// TwinCAT 3 PLC project SlitterPlc
// ProgramVersion: 3.1.4023.0
// libraries:
//   Tc2_Math, * (Beckhoff Automation GmbH)
//   Tc2_MC2, * (Beckhoff Automation GmbH)
//   Tc2_ModbusSrv, * (Beckhoff Automation GmbH)
//   Tc2_Standard, * (Beckhoff Automation GmbH)
//   Tc2_System, * (Beckhoff Automation GmbH)
//   Tc2_Utilities, * (Beckhoff Automation GmbH)
//   Tc2_XmlDataSrv, * (Beckhoff Automation GmbH)
//   Tc3_EventLogger, * (Beckhoff Automation GmbH)
//   Tc3_Module, * (Beckhoff Automation GmbH)
//   Tc3_PackML_V2, * (Beckhoff Automation GmbH)
//   VisuDialogs, * (System)
// project tree:
//   DUTs/Parameters/ ST_CameraParameters.TcDUT, ST_CutterParameters.TcDUT, ST_EjectorParameters.TcDUT, ST_MandrelParameters.TcDUT
//   DUTs/ ST_CameraData.TcDUT, ST_CameraResults.TcDUT, ST_InspectCommands.TcDUT, ST_ManualCommands.TcDUT, ST_TubeParameters.TcDUT
//   Ellipse/ FB_ComputeFromImage.TcPOU, FB_Ellipse.TcPOU, FB_FourthOrder.TcPOU, FB_SecondOrder.TcPOU
//   / GlobalTextList.TcGTLO, PlcTask.TcTTO, Visualization Manager.TcVMO (not stored), VISU_TASK.TcTTO
//   GVLs/ GVL.TcGVL
//   ITFs/ I_Actuator.TcIO, I_Axis.TcIO, I_Camera.TcIO, I_Frame.TcIO
//   POUs/ FB_Actuator.TcPOU, FB_Axis.TcPOU, FB_Base.TcPOU, FB_Camera.TcPOU, FB_Cutter.TcPOU, FB_Ejector.TcPOU, FB_Frame.TcPOU, FB_Mandrel.TcPOU, FB_Slitter.TcPOU, MAIN.TcPOU
//   VISUs/ Front_Panel.TcVIS, Manual_Inspect.TcVIS, MachineSettings.TcVIS, ManualControl.TcVIS, Manual_Camera.TcVIS, Manual_Camera_Calibration.TcVIS, Manual_Camera_Inspection.TcVIS, Manual_Camera_Inspection_Raw.TcVIS, Manual_Camera_RawData.TcVIS, Manual_Cutter.TcVIS, Manual_Ejector.TcVIS, Manual_Frame.TcVIS, Manual_Mandrel.TcVIS, Manual_Vacuum.TcVIS, Manual_Select_Tube.TcVIS, Settings.TcVIS, SettingsTemplate.TcVIS, Settings_Mandrel.TcVIS, Settings_PassCriteria.TcVIS, Settings_ProductDimensions.TcVIS, Visualization.TcVIS

CONFIGURATION SlitterPlc
    RESOURCE PLC ON TwinCAT3
        TASK PlcTask(INTERVAL := T#10ms, PRIORITY := 20);
        TASK VISU_TASK(INTERVAL := T#200000us, PRIORITY := 30);
        PROGRAM MAIN WITH PlcTask : MAIN;
        PROGRAM VisuElems_Visu_Prg WITH VISU_TASK : VisuElems.Visu_Prg;
    END_RESOURCE
END_CONFIGURATION

// ---- DUTs/Parameters/ST_CameraParameters.TcDUT
TYPE ST_CameraParameters :
STRUCT
	pitchRow	: LREAL; // := 0.0250;
	pitchColumn	: LREAL; //  := 0.0219;
	calibrationDistance	: LREAL; // := 3;
	angle		: LREAL; // := 27.65;
END_STRUCT
END_TYPE

// ---- DUTs/Parameters/ST_CutterParameters.TcDUT
TYPE ST_CutterParameters :
STRUCT
	retractPosition	: LREAL; // := 10;
	cutVelocity	: LREAL; // := 20;
END_STRUCT
END_TYPE

// ---- DUTs/Parameters/ST_EjectorParameters.TcDUT
TYPE ST_EjectorParameters :
STRUCT
	ejectPositionPass 	: LREAL; // := 100;
	ejectPositionHome 	: LREAL; // := 50;
	ejectPositionFail 	: LREAL; // := 0;
	ejectVelocity		: LREAL; // := 20;
END_STRUCT
END_TYPE

// ---- DUTs/Parameters/ST_MandrelParameters.TcDUT
TYPE ST_MandrelParameters :
STRUCT
	loadPositionX	: LREAL; // := -72.5;
	velocityX		: LREAL; // := 10;
	loadPositionY	: LREAL; // := -22;
	velocityY		: LREAL; // := 250;
	spindleVelocity	: LREAL; // := 20;
	spindleOffset	: LREAL; // := -1;
	vacuumVelocity	: LREAL; // := 360;
END_STRUCT
END_TYPE

// ---- DUTs/ST_CameraData.TcDUT
TYPE ST_CameraData :
STRUCT
	CurrentJobID			: WORD;
	ErrorCode				: WORD;
	AcquisitionID			: WORD;
	InspectionID			: WORD;
	InspectionResultCode	: WORD;
	Results					: ST_CameraResults;
END_STRUCT
END_TYPE

// ---- DUTs/ST_CameraResults.TcDUT
TYPE ST_CameraResults :
STRUCT
	Count				: REAL;
	WidthMeasurement	: REAL;
	HeightMeasurement	: REAL;
	LocationInX			: REAL;
	LocationInY			: REAL;
	PatternMatchRow		: REAL;
	PatternMatchColumn 	: REAL;
	PointValueRow		: ARRAY[1..GVL.NumberVisionPoints] OF REAL;
	PointValueColumn	: ARRAY[1..GVL.NumberVisionPoints] OF REAL;
END_STRUCT
END_TYPE

// ---- DUTs/ST_InspectCommands.TcDUT
TYPE ST_InspectCommands :
STRUCT
	IncrementSpindle 	: BOOL;
	DecrementSpindle	: BOOL;
	Inspect				: BOOL;	
	InspectComplete		: BOOL;
END_STRUCT
END_TYPE

// ---- DUTs/ST_ManualCommands.TcDUT
TYPE ST_ManualCommands :
STRUCT
	bCalibrateMandrel		: BOOL;
	bCameraCalibrate		: BOOL;
	bCameraComputePeak		: BOOL;
	bCameraTrigger			: BOOL;
	bCameraInspect			: BOOL;
	bCameraRawData			: BOOL;
	bCameraSelectTube		: BOOL;
	bCutSample				: BOOL;
	bCutterDisable			: BOOL;
	bCutterHome				: BOOL;
	bCutterReset			: BOOL;
	bCutterMoveAbs			: BOOL;
	bEjectAxisEnableToggle	: BOOL;
	bEjectAxisFailPosition	: BOOL;
	bEjectAxisHomePosition	: BOOL;
	bEjectAxisPassPosition	: BOOL;
	bEjectAxisReset			: BOOL;
	bEjectReset				: BOOL;
	bEjectSamplePass		: BOOL;
	bEjectSampleFail		: BOOL;
	bEjectZExtend			: BOOL;
	bEjectZNeutral			: BOOL;
	bEjectZRetract			: BOOL;
	bEjectBlowOff			: BOOL;
	bEjectVacuum			: BOOL;
	bEjectXOff				: BOOL;
	bEjectZOff				: BOOL;
	bLowerMandrel			: BOOL;		
	bMandrelXEnableToggle	: BOOL;
	bMandrelYEnableToggle	: BOOL;
	bMandrelSpindleToggle	: BOOL;
	bMandrelSpindleRotate	: BOOL;
	bMandrelReset			: BOOL;
	bMoveToLoadPosition		: BOOL;
	bMoveToCutPosition		: BOOL;
	bMoveToEjectPosition	: BOOL;
	bMoveToInspectPosition	: BOOL;
	bRaiseMandrel			: BOOL;
	bSaveMandrelParameters	: BOOL;
	bToggleMandrelVacuum	: BOOL;
	bVacuumAxisToggleEnable	: BOOL;
	bVacuumAxisMove			: BOOL;
	bVacuumAxisReset		: BOOL;
END_STRUCT
END_TYPE

// ---- DUTs/ST_TubeParameters.TcDUT
TYPE ST_TubeParameters :
STRUCT
	Index				: INT;
	Description			: STRING;
	ProductName			: STRING;
	Diameter			: LREAL;	// diameter [mm] of tube at top protrusion
	DepthOfPocket		: LREAL;	// cut surface offset from top most surface [mm]
	MinLength			: LREAL;	// criteria: minimum length of an allowable cut length [mm]
	MaxLength			: LREAL;	// criteria: maximum length of an allowable cut length [mm]
	MinHeight			: LREAL;	// criteria: minimum width of blob of cut [mm]
	MaxHeight			: LREAL;	// criteria: maximum width of blob of cut [mm]
	ResultToleranceX	: LREAL;	// criteria: allowable difference from center of tube to center of cut x axis
	ResultToleranceY	: LREAL;	// criteria: allowable difference from center of tube to center of cut y axis
	AdjustmentX			: LREAL;  	// adjustment to add to result in mm before determining pass/fail
	AdjustmentY			: LREAL;	// adjustment to add to result in mm before determining pass/fail
	AdjustmentLength	: LREAL;	// adjustment to add to length result in mm before determining pass/fail	
	CutPositionX		: LREAL;	
	CutPositionY		: LREAL;
	InspectPositionX 	: LREAL;
	InspectPositionY 	: LREAL;
	EjectPositionX		: LREAL;
	EjectPositionY		: LREAL;
	VacPosition			: LREAL;	// vacuum axis position
	VacuumThreshold		: REAL; 	// mmHg to detect presence of tube on mandrel	
	ComputerProgram		: STRING := 'Tube';
END_STRUCT
END_TYPE

// ---- GVLs/GVL.TcGVL
{attribute 'qualified_only'}
VAR_GLOBAL CONSTANT
	NumberVisionPoints	: INT := 20;	// number of points from the camera vision system
	NumberEllipsePoints	: INT := 40; 	// number of ellipse points is 2x number of vision points
	Unknowns			: INT := 5;		// ellipse coefficients
	MaxIterations		: INT := 50;	
	ConvergenceCriteria : LREAL := 0.000000001;	
	CameraIpAddress		: STRING := '192.168.1.2';
	ModbusReadOffset	: WORD := 7000;
	ModbusWriteOffset	: WORD := 2000;
END_VAR

// ---- ITFs/I_Actuator.TcIO
INTERFACE I_Actuator

PROPERTY Error : BOOL
GET
END_GET
SET
END_SET
END_PROPERTY

METHOD Extend : INT
VAR_INPUT
END_VAR
END_METHOD

PROPERTY IsExtended : BOOL
GET
END_GET
END_PROPERTY

PROPERTY IsRetracted : BOOL
GET
END_GET
END_PROPERTY

METHOD Neutral : BOOL
VAR_INPUT
END_VAR
END_METHOD

METHOD Retract : INT
VAR_INPUT
END_VAR
END_METHOD

END_INTERFACE

// ---- ITFs/I_Axis.TcIO
INTERFACE I_Axis

PROPERTY ErrorCode : UDINT
GET
END_GET
END_PROPERTY

METHOD Home : INT
VAR_INPUT
	Execute	: BOOL;
END_VAR
END_METHOD

METHOD MoveAbs : INT
VAR_INPUT
	Execute	: BOOL;
END_VAR
END_METHOD

METHOD MoveRel : INT
VAR_INPUT
	Execute	: BOOL;
END_VAR
END_METHOD

PROPERTY NcToPlc : NCTOPLC_AXIS_REF
GET
END_GET
END_PROPERTY

METHOD Power : BOOL
VAR_INPUT
	Enable	: BOOL;
END_VAR
END_METHOD

METHOD Reset : INT
VAR_INPUT
	Execute	: BOOL;
END_VAR
END_METHOD

PROPERTY SetDistance : LREAL
SET
END_SET
END_PROPERTY

PROPERTY SetPosition : LREAL
SET
END_SET
END_PROPERTY

PROPERTY SetVelocity : LREAL
SET
END_SET
END_PROPERTY

PROPERTY Status : ST_AxisStatus
GET
END_GET
END_PROPERTY

END_INTERFACE

// ---- ITFs/I_Camera.TcIO
INTERFACE I_Camera

METHOD Calibrate : BOOL
VAR_INPUT
END_VAR
END_METHOD

PROPERTY CalibrationDistance : LREAL
GET
END_GET
SET
END_SET
END_PROPERTY

PROPERTY CameraProgram : STRING
GET
END_GET
SET
END_SET
END_PROPERTY

METHOD Compute : INT
VAR_INPUT
	Execute		: BOOL;	
END_VAR
END_METHOD

PROPERTY CutLengthWithOffset : REAL
GET
END_GET
SET
END_SET
END_PROPERTY

PROPERTY DeltaXmmWithOffset : REAL
GET
END_GET
SET
END_SET
END_PROPERTY

PROPERTY DeltaYmmWithOffset : REAL
GET
END_GET
SET
END_SET
END_PROPERTY

PROPERTY Fail : BOOL
GET
END_GET
SET
END_SET
END_PROPERTY

METHOD GetCameraData : INT
VAR_INPUT
END_VAR
END_METHOD

METHOD Inspect : INT
VAR_INPUT
	Execute	: BOOL;
END_VAR
END_METHOD

END_INTERFACE

// ---- ITFs/I_Frame.TcIO
INTERFACE I_Frame

METHOD BlinkGreen : BOOL
VAR_INPUT
END_VAR
END_METHOD

PROPERTY ControlLeft : BOOL
GET
END_GET
END_PROPERTY

PROPERTY ControlRight : BOOL
GET
END_GET
END_PROPERTY

PROPERTY Door1 : BOOL
GET
END_GET
END_PROPERTY

PROPERTY Door2 : BOOL
GET
END_GET
END_PROPERTY

PROPERTY Door3 : BOOL
GET
END_GET
END_PROPERTY

PROPERTY GreenLight : BOOL
GET
END_GET
SET
END_SET
END_PROPERTY

END_INTERFACE

// ---- POUs/MAIN.TcPOU
PROGRAM MAIN
VAR PERSISTENT
	TubeSelection		: ARRAY[1..5] OF ST_TubeParameters; // array of tube parameters saved in memory
END_VAR
VAR
	CutOffValve	AT %Q*	: BOOL;
	Tube				: ST_TubeParameters;		// parameters in use by the machine
	TubeHmi				: ST_TubeParameters;		// parameters to edit in the hmi
	
	TubeIndicator		: ARRAY[1..5] OF BOOL := [TRUE, FALSE, FALSE, FALSE, FALSE];		// indicator as to which tube is in use
	
	fbSlitter			: FB_Slitter;				// object of machine
	Frame				: FB_Frame;	
	eCommand			: Tc3_PackML_V2.E_PMLCommand;
	eModeCommand		: DINT := E_PMLProtectedUnitMode.ePMLProtUnitMode_Production;
	eState				: Tc3_PackML_V2.E_PMLState;
	sState				: STRING;
	eMode				: DINT;

	TONhmi				: TON;
	TONidle				: TON := (PT := T#2M);
	ntStartProcess		: NT_StartProcess;

	bSave				: BOOL;
	bProcessing			: BOOL;
	bFailed				: BOOL;
	bPassed				: BOOL;
	fbWritePersistent	: FB_WritePersistentData;

	i					: INT;
	
	bOperation			: BOOL;
	bManual				: BOOL;
	bProductSettings	: BOOL;
	bMachineSettings	: BOOL;
	hmiStatus			: STRING := 'OK';
	PressureOn			: BOOL;
	PressureOnTon		: TON := (PT := T#10S);
	PressureOffTon		: TON := (PT := T#2s);
	hmiReset			: BOOL;
	bInspect			: BOOL;
	bNoDetect			: BOOL;
	InspectCommands		: ST_InspectCommands;
	
	currentUser: WSTRING;
	actualCurrentUser: WSTRING;
	debug1			: INT;
	debug2			: INT;
	nIndex			: INT;
	j				: INT;
	readTubeParameter	: ST_TubeParameters;
	emptyTubeParameter	: ST_TubeParameters;
	FilesLoaded		: BOOL;
	rTrigWriteFiles	: R_TRIG;
	nWriteFiles		: INT;
	fbXmlSrvRead	: FB_XmlSrvRead;
	fbXmlSrvWrite	: FB_XmlSrvWrite;
	fbMessage		: FB_TcMessage;
	x : INT;
END_VAR
VAR PERSISTENT	
	iBatch				: ULINT;
	iCounter			: ULINT;
	iCountFailed		: UINT;
	hmiBatch			: ULINT;
	CycleCounter		: LREAL;
END_VAR

CutOffValve := TRUE;

// set up the event logger message
IF NOT fbMessage.EqualsToEventEntryEx(stOther := TC_EVENTS.SlitterEvents.TubeParameterChange) THEN
	fbMessage.CreateEx(TC_EVENTS.SlitterEvents.TubeParameterChange, 0);
	fbMessage.ipArguments.Clear();
END_IF

// load the config parameters on start up
A_ReadTubeParameters();

// display the current user
IF currentUser <> VisuElems.CurrentFullUserName THEN
	currentUser := VisuElems.CurrentFullUserName;
END_IF

IF bOperation THEN				// when switching to the Operation page
	bOperation := FALSE;
	FOR i:=1 TO 5 DO
		TubeIndicator[i] := FALSE;
	END_FOR
	TubeIndicator[1] := TRUE;
	Tube := TubeSelection[1];	// set the tube selection to the first tube on entering page
	TubeHmi := Tube;			// write the parameters to the HMI display
END_IF

IF bManual THEN
	bManual := FALSE;
	TubeHmi := Tube;	// write the parameters to the HMI display
						// do not change the selected tube
END_IF

IF bProductSettings THEN
	bProductSettings := FALSE;
	FOR i:=1 TO 5 DO
		TubeIndicator[i] := FALSE;
	END_FOR
	TubeIndicator[1] := TRUE;
	Tube := TubeSelection[1];	// on entering product page select the first tube
	TubeHmi := Tube;			// write the parameters to the HMI display
END_IF

IF bMachineSettings THEN
	bMachineSettings := FALSE;
	TubeHmi := Tube;
END_IF

//A_StartVisualization();
A_PackMlCommands();

// this must be called before the fbSlitter execution
// determines the tube that is selected 
FOR i := 1 TO 5 DO
	IF TubeIndicator[i] THEN
		Tube := TubeSelection[i];
	END_IF
END_FOR

// machine object
fbSlitter(
	eCommand := eCommand,
	eModeCommand := eModeCommand,
	Batch := hmiBatch,
	Tube := Tube,
	TubeHmi := TubeHmi,	// used only for manual commands
	Inspect := bInspect,
	InspectCmd := InspectCommands,
	CounterOut => iCounter,
	CountFailedOut => iCountFailed,
	BatchOut => iBatch,
	eState => eState,
	sState => sState,
	eMode => eMode);

IF eState <> E_PMLState.ePMLState_Undefined THEN
	A_MonitorParameters();
	A_WriteParameters();
END_IF	
A_StatusIndicator();
(*		
FOR i := 1 TO 5 DO
	IF TubeIndicator[i] THEN
		debug2 := debug2 + 1;		
		IF MEMCMP(ADR(Tube), ADR(TubeSelection[i]), SIZEOF(tube)) <> 0 THEN
			TubeHmi := Tube;		
			bSave := TRUE;
			debug1 := debug1 + 1;
		END_IF 
	END_IF
END_FOR
*)

ACTION A_MonitorParameters:
IF MEMCMP(ADR(TubeHmi), ADR(TubeSelection[i]), SIZEOF(TubeHmi)) <> 0 THEN
	IF TubeHmi.AdjustmentLength <> TubeSelection[i].AdjustmentLength THEN
		// Tube {0} Parameter {1} changed from {2} to {3}
		fbMessage.ipArguments.Clear();
		fbMessage.ipArguments.AddInt(i).AddString('AdjustmentLength');
		fbMessage.ipArguments.AddLReal(TubeSelection[i].AdjustmentLength).AddLReal(TubeHmi.AdjustmentLength);
		fbMessage.Send(0);
	END_IF
	IF TubeHmi.AdjustmentX <> TubeSelection[i].AdjustmentX THEN
		fbMessage.ipArguments.Clear();
		fbMessage.ipArguments.AddInt(i).AddString('AdjustmentX');
		fbMessage.ipArguments.AddLReal(TubeSelection[i].AdjustmentX).AddLReal(TubeHmi.AdjustmentX);
		fbMessage.Send(0);				
	END_IF
	IF TubeHmi.AdjustmentY <> TubeSelection[i].AdjustmentY THEN
		fbMessage.ipArguments.Clear();
		fbMessage.ipArguments.AddInt(i).AddString('AdjustmentY');
		fbMessage.ipArguments.AddLReal(TubeSelection[i].AdjustmentY).AddLReal(TubeHmi.AdjustmentY);
		fbMessage.Send(0);								
	END_IF
	IF TubeHmi.CutPositionX <> TubeSelection[i].CutPositionX THEN
		fbMessage.ipArguments.Clear();
		fbMessage.ipArguments.AddInt(i).AddString('CutPositionX');
		fbMessage.ipArguments.AddLReal(TubeSelection[i].CutPositionX).AddLReal(TubeHmi.CutPositionX);
		fbMessage.Send(0);												
	END_IF
	IF TubeHmi.CutPositionY <> TubeSelection[i].CutPositionY THEN
		fbMessage.ipArguments.Clear();
		fbMessage.ipArguments.AddInt(i).AddString('CutPositionY');
		fbMessage.ipArguments.AddLReal(TubeSelection[i].CutPositionY).AddLReal(TubeHmi.CutPositionY);
		fbMessage.Send(0);																
	END_IF
	IF TubeHmi.DepthOfPocket <> TubeSelection[i].DepthOfPocket THEN
		fbMessage.ipArguments.Clear();
		fbMessage.ipArguments.AddInt(i).AddString('DepthOfPocket');
		fbMessage.ipArguments.AddLReal(TubeSelection[i].DepthOfPocket).AddLReal(TubeHmi.DepthOfPocket);
		fbMessage.Send(0);																				
	END_IF
	IF TubeHmi.Description <> TubeSelection[i].Description THEN
		fbMessage.ipArguments.Clear();
		fbMessage.ipArguments.AddInt(i).AddString('Description');
		fbMessage.ipArguments.AddString(TubeSelection[i].Description).AddStringByValue(TubeHmi.Description);
		fbMessage.Send(0);																								
	END_IF
	IF TubeHmi.Diameter <> TubeSelection[i].Diameter THEN
		fbMessage.ipArguments.Clear();
		fbMessage.ipArguments.AddInt(i).AddString('Diameter');
		fbMessage.ipArguments.AddLReal(TubeSelection[i].Diameter).AddLReal(TubeHmi.Diameter);
		fbMessage.Send(0);																												
	END_IF
	IF TubeHmi.EjectPositionX <> TubeSelection[i].EjectPositionX THEN
		fbMessage.ipArguments.Clear();
		fbMessage.ipArguments.AddInt(i).AddString('EjectPositionX');
		fbMessage.ipArguments.AddLReal(TubeSelection[i].EjectPositionX).AddLReal(TubeHmi.EjectPositionX);
		fbMessage.Send(0);																												
	END_IF	
	IF TubeHmi.EjectPositionY <> TubeSelection[i].EjectPositionY THEN
		fbMessage.ipArguments.Clear();
		fbMessage.ipArguments.AddInt(i).AddString('EjectPositionY');
		fbMessage.ipArguments.AddLReal(TubeSelection[i].EjectPositionY).AddLReal(TubeHmi.EjectPositionY);
		fbMessage.Send(0);																												
	END_IF
	IF TubeHmi.InspectPositionX <> TubeSelection[i].InspectPositionX THEN
		fbMessage.ipArguments.Clear();
		fbMessage.ipArguments.AddInt(i).AddString('InspectPositionX');
		fbMessage.ipArguments.AddLReal(TubeSelection[i].InspectPositionX).AddLReal(TubeHmi.InspectPositionX);
		fbMessage.Send(0);																																
	END_IF
	IF TubeHmi.InspectPositionY <> TubeSelection[i].InspectPositionY THEN
		fbMessage.ipArguments.Clear();
		fbMessage.ipArguments.AddInt(i).AddString('InspectPositionY');
		fbMessage.ipArguments.AddLReal(TubeSelection[i].InspectPositionY).AddLReal(TubeHmi.InspectPositionY);
		fbMessage.Send(0);																																				
	END_IF
	IF TubeHmi.MaxHeight <> TubeSelection[i].MaxHeight THEN
		fbMessage.ipArguments.Clear();
		fbMessage.ipArguments.AddInt(i).AddString('MaxHeight');
		fbMessage.ipArguments.AddLReal(TubeSelection[i].MaxHeight).AddLReal(TubeHmi.MaxHeight);
		fbMessage.Send(0);																																								
	END_IF
	IF TubeHmi.MaxLength <> TubeSelection[i].MaxLength THEN
		fbMessage.ipArguments.Clear();
		fbMessage.ipArguments.AddInt(i).AddString('MaxLength');
		fbMessage.ipArguments.AddLReal(TubeSelection[i].MaxLength).AddLReal(TubeHmi.MaxLength);
		fbMessage.Send(0);																																												
	END_IF
	IF TubeHmi.MinHeight <> TubeSelection[i].MinHeight THEN
		fbMessage.ipArguments.Clear();
		fbMessage.ipArguments.AddInt(i).AddString('MinHeight');
		fbMessage.ipArguments.AddLReal(TubeSelection[i].MinHeight).AddLReal(TubeHmi.MinHeight);
		fbMessage.Send(0);																																																
	END_IF
	IF TubeHmi.MinLength <> TubeSelection[i].MinLength THEN
		fbMessage.ipArguments.Clear();
		fbMessage.ipArguments.AddInt(i).AddString('MinLength');
		fbMessage.ipArguments.AddLReal(TubeSelection[i].MinLength).AddLReal(TubeHmi.MinLength);
		fbMessage.Send(0);																																																				
	END_IF
	IF TubeHmi.ProductName <> TubeSelection[i].ProductName THEN
		fbMessage.ipArguments.Clear();
		fbMessage.ipArguments.AddInt(i).AddString('ProductName');
		fbMessage.ipArguments.AddString(TubeSelection[i].ProductName).AddString(TubeHmi.ProductName);
		fbMessage.Send(0);																																																				
	END_IF
	IF TubeHmi.ResultToleranceX <> TubeSelection[i].ResultToleranceX THEN
		fbMessage.ipArguments.Clear();
		fbMessage.ipArguments.AddInt(i).AddString('ResultToleranceX');
		fbMessage.ipArguments.AddLReal(TubeSelection[i].ResultToleranceX).AddLReal(TubeHmi.ResultToleranceX);
		fbMessage.Send(0);																																																				
	END_IF
	IF TubeHmi.ResultToleranceY <> TubeSelection[i].ResultToleranceY THEN
		fbMessage.ipArguments.Clear();
		fbMessage.ipArguments.AddInt(i).AddString('ResultToleranceY');
		fbMessage.ipArguments.AddLReal(TubeSelection[i].ResultToleranceY).AddLReal(TubeHmi.ResultToleranceY);
		fbMessage.Send(0);																																																								
	END_IF
	IF TubeHmi.VacuumThreshold <> TubeSelection[i].VacuumThreshold THEN
		fbMessage.ipArguments.Clear();
		fbMessage.ipArguments.AddInt(i).AddString('VacuumThreshold');
		fbMessage.ipArguments.AddLReal(TubeSelection[i].VacuumThreshold).AddLReal(TubeHmi.VacuumThreshold);
		fbMessage.Send(0);																																																								
	END_IF
END_IF
END_ACTION

ACTION A_PackMlCommands:
PressureOffTon(IN := frame.Pressure < 80);
IF PressureOffTon.Q THEN
	PressureOn := FALSE;
END_IF
PressureOnTON(IN := frame.Pressure > 80);
IF PressureOnTON.Q THEN
	PressureOn := TRUE;
END_IF

// pack ml commands
IF (NOT PressureOn OR hmiReset) AND FilesLoaded THEN
 	eCommand := E_PMLCommand.ePMLCommand_Abort;
	hmiReset := FALSE;
	IF NOT PressureOn THEN
		hmiStatus := 'Pressure<80PSIG';
	END_IF
ELSIF eMode = E_PMLProtectedUnitMode.ePMLProtUnitMode_Manual THEN
	hmiStatus := 'Manual Mode';
	IF eModeCommand = E_PMLProtectedUnitMode.ePMLProtUnitMode_Production THEN
		eCommand := E_PMLCommand.ePMLCommand_Abort;
		Frame.GreenLight := FALSE;
	ELSE
		CASE eState OF
			E_PMLState.ePMLState_Undefined: eCommand := E_PMLCommand.ePMLCommand_Abort;
			E_PMLState.ePMLState_Aborted: eCommand := E_PMLCommand.ePMLCommand_Clear;
			E_PMLState.ePMLState_Idle: eCommand := E_PMLCommand.ePMLCommand_Start;
			E_PMLState.ePMLState_Stopped: eCommand := E_PMLCommand.ePMLCommand_Reset;
			E_PMLState.ePMLState_Aborting: eCommand := E_PMLCommand.ePMLCommand_Undefined;
		END_CASE
	END_IF
ELSIF eMode = E_PMLProtectedUnitMode.ePMLProtUnitMode_Production THEN
	hmiStatus := 'Automatic Mode';
	IF eModeCommand = E_PMLProtectedUnitMode.ePMLProtUnitMode_Manual THEN
		eCommand := E_PMLCommand.ePMLCommand_Abort;
	ELSE
		CASE eState OF
			E_PMLState.ePMLState_Undefined:
				IF FilesLoaded THEN
					eCommand := E_PMLCommand.ePMLCommand_Abort;
				END_IF
			E_PMLState.ePMLState_Aborted:  
				//IF NOT Frame.Door1 AND NOT Frame.Door2 THEN
					eCommand := E_PMLCommand.ePMLCommand_Clear;
				//END_IF
			E_PMLState.ePMLState_Idle:
					Frame.GreenLight := Frame.Door1 AND Frame.Door2 AND Frame.Door3 AND Frame.Door4;
					IF Frame.GreenLight THEN
						hmiStatus := 'Ready';
					ELSE
						hmiStatus := 'Door Open';
					END_IF
					IF (Frame.ControlLeft AND Frame.ControlRight) AND Frame.GreenLight THEN
						eCommand := E_PMLCommand.ePMLCommand_Start;
						Frame.GreenLight := FALSE;
					END_IF
			E_PMLState.ePMLState_Complete: eCommand := E_PMLCommand.ePMLCommand_Reset;
														
			E_PMLState.ePMLState_Stopped: eCommand := E_PMLCommand.ePMLCommand_Reset;
			E_PMLState.ePMLState_Aborting: eCommand := E_PMLCommand.ePMLCommand_Undefined;			
		END_CASE
	END_IF
END_IF
END_ACTION

ACTION A_ReadTubeParameters:
x := x + 1;

CASE nIndex OF
	0: // read the info from the config file for the camera
		j := 1;
		nIndex := 10;
	10: // 
		fbXmlSrvRead.sXPath := CONCAT('/Configuration/TubeParameters/Tube', INT_TO_STRING(j));
		fbXmlSrvRead.pSymAddr := ADR(readTubeParameter);
		fbXmlSrvRead.cbSymSize := SIZEOF(readTubeParameter);
		fbXmlSrvRead.bExecute := TRUE;
		nIndex := 20;
	20: // wait for the info to load
		IF NOT fbXmlSrvRead.bBusy THEN
			fbXmlSrvRead.bExecute := FALSE;
			MEMCPY(ADR(TubeSelection[j]), ADR(readTubeParameter), SIZEOF(readTubeParameter));
			MEMCPY(ADR(readTubeParameter), ADR(emptyTubeParameter), SIZEOF(emptyTubeParameter));
			nIndex := 30;
			IF j >= 5 THEN
				nIndex := 30;
			ELSE
				nIndex := 10;
				j := j + 1;
			END_IF
		END_IF
	30: // set variables
		Tube := TubeSelection[1];
		TubeHmi := TubeSelection[1];
		TubeIndicator[1] := TRUE;
		bProcessing := FALSE;
		bPassed := FALSE;
		bFailed := FALSE;
		bNoDetect := FALSE;
		nIndex := 40;
	40: // wait here for files loaded
		IF fbSlitter.ReadParameters(Execute := TRUE) THEN
			fbSlitter.ReadParameters(Execute := FALSE);
			FilesLoaded := TRUE;
			nIndex := 50;
		END_IF
	50: // 
		
END_CASE

fbXmlSrvRead(
	sNetId:= '', 
	ePath:= E_OpenPath.PATH_GENERIC, 
	nMode:= XMLSRV_SKIPMISSING, 
	sFilePath:= 'C:\Configuration.xml');
END_ACTION

ACTION A_StartVisualization:
// start the hmi

TONhmi(IN := TRUE, PT := T#4S);
IF TONhmi.Q THEN
	ntStartProcess(
		NETID := '',
		PATHSTR := 'C:\TwinCAT\3.1\Components\Plc\Tc3PlcHmi\Tc3PlcHmi.exe',
		DIRNAME := 'C:\TwinCAT\3.1\Components\Plc\Tc3PlcHmi\',
		COMNDLINE := 'Tc3PlcHmi.exe',
		START := TRUE);
END_IF
END_ACTION

ACTION A_StatusIndicator:
// status indicator

IF eMode = E_PMLProtectedUnitMode.ePMLProtUnitMode_Production THEN
	CASE fbSlitter.Status OF
		0: // idle if idle is on for more than 2 minutes, remove the result
			TONidle(IN := TRUE);
			bProcessing := FALSE;
			IF TONidle.Q THEN
				bFailed := FALSE;
				bPassed := FALSE;	
				bNoDetect := FALSE;		
			END_IF
		1: // processing
			bProcessing := TRUE;
			bFailed := FALSE;
			bPassed := FALSE;
			bNoDetect := FALSE;
			TONidle(IN := FALSE);
		2: // pass
			bPassed := TRUE;
			bFailed := FALSE;
			bProcessing := FALSE;
			bNoDetect := FALSE;
		3: // fail	
			bPassed := FALSE;
			bFailed := TRUE;
			bProcessing := FALSE;
			bNoDetect := FALSE;
		4: // failed to detect
			bPassed := FALSE;
			bFailed := FALSE;
			bProcessing := FALSE;
			bNoDetect := TRUE;		
	END_CASE
ELSE
	bPassed := FALSE;
	bFailed := FALSE;
	bProcessing := FALSE;
END_IF
END_ACTION

ACTION A_WriteParameters:
// write persistent data 
rTrigWriteFiles(CLK := bSave);
IF rTrigWriteFiles.Q THEN
	fbSlitter.SaveParameters(Execute := FALSE);
	nWriteFiles := 10;
END_IF

IF NOT bSave THEN
	nWriteFiles := 0;
END_IF

CASE nWriteFiles OF
	10: // get the tube into memory
		FOR i := 1 TO 5 DO
			IF TubeIndicator[i] THEN
				A_MonitorParameters();
				TubeSelection[i] := TubeHmi;
				TubeSelection[i].Index := i;
			END_IF
		END_FOR
		j := 1;
		nWriteFiles := 20;
	20: // write the tube parameters
		MEMCPY(ADR(readTubeParameter), ADR(TubeSelection[j]), SIZEOF(readTubeParameter));
		fbXmlSrvWrite.bExecute := TRUE;
		fbXmlSrvWrite.cbSymSize := SIZEOF(readTubeParameter);
		fbXmlSrvWrite.pSymAddr := ADR(readTubeParameter);
		fbXmlSrvWrite.sXPath := CONCAT('/Configuration/TubeParameters/Tube', INT_TO_STRING(j));
		nWriteFiles := 30;
	30: // wait to complete
		IF NOT fbXmlSrvWrite.bBusy THEN
			fbXmlSrvWrite.bExecute := FALSE;
			IF j >= 5 THEN
				nWriteFiles := 40;
			ELSE
				j := j + 1;
				nWriteFiles := 20;
			END_IF
		END_IF
	40: // command slitter to save parameters
		IF fbSlitter.SaveParameters(Execute := TRUE) THEN
			fbSlitter.SaveParameters(Execute := FALSE);
			nWriteFiles := 50;
		END_IF
	50: // done state
		bSave := FALSE;
END_CASE

fbXmlSrvWrite(
	sNetId:= '', 
	ePath:= E_OpenPath.PATH_GENERIC, 
	nMode:= XMLSRV_SKIPMISSING, 
	sFilePath:= 'C:\Configuration.xml');
END_ACTION

END_PROGRAM

// ---- POUs/FB_Slitter.TcPOU
FUNCTION_BLOCK FB_Slitter EXTENDS FB_BASE IMPLEMENTS I_UnitState
VAR_INPUT
	Batch		: ULINT;
	Inspect		: BOOL;					// run routine without cut; just inspect
	InspectCmd	: ST_InspectCommands;
	TubeHmi		: ST_TubeParameters;	// used for manual commands
END_VAR
VAR_IN_OUT
	Tube		: ST_TubeParameters;
END_VAR
VAR_OUTPUT 
	FilesLoaded		: BOOL;
	BatchOut		: ULINT;
	CounterOut		: ULINT;
	CountFailedOut	: UINT;
	Status			: INT; 	// 0 = idle, 1 = processing, 2 = pass, 3 = fail, 4 = no detect
END_VAR
VAR
	Mandrel				: FB_Mandrel;
	MandrelParameters	: ST_MandrelParameters;
	Camera				: FB_Camera;
	CameraParameters	: ST_CameraParameters;
	Cutter				: FB_Cutter;
	CutterParameters 	: ST_CutterParameters;
	Ejector				: FB_Ejector;
	EjectorParameters	: ST_EjectorParameters;
	EjectState			: INT;
	Eject				: BOOL;
	
	Manual		: ST_ManualCommands;
	bBusy		: BOOL;	
	bCalibration: BOOL;
	strJobName	: STRING;	// for manual override of which camera program is used
	nIndex		: INT;
	PreviousTubeIndex	: INT;
	fbFileOpen	: FB_FileOpen;
	fbFileWrite	: FB_FileWrite;
	fbFileClose	: FB_FileClose;
	fbLocalSystemTime	: FB_LocalSystemTime;
	bDecrementSpindle: BOOL;
	bIncrementSpindle: BOOL;
	bInspect: BOOL;
	bInspectComplete: BOOL;
	nCalibrationCounter : INT;
	CalibrationArrayX	: ARRAY[0..CalMax] OF LREAL;
	CalibrationArrayY	: ARRAY[0..CalMax] OF LREAL;
	AverageX 			: LREAL;
	AverageY 			: LREAL;
	
	fbXmlSrvRead		: FB_XmlSrvRead;
	fbXmlSrvWrite		: FB_XmlSrvWrite;

	fbMessageSaved		: FB_TcMessage;
		
END_VAR
VAR CONSTANT
	CalMax	: INT := 9;
END_VAR
VAR PERSISTENT
	Counter		: UINT;
	CountFailed	: UINT;
END_VAR


SUPER^();

IF eState <> E_PMLState.ePMLState_Undefined THEN
	Mandrel.MonitorParameters();
	Camera.MonitorParameters();
	Cutter.MonitorParameters();
	Ejector.MonitorParameters();
END_IF

Mandrel.ConvertVaccum();
Mandrel.TubeParameters := Tube;

IF Batch <> BatchOut THEN
	BatchOut := Batch;
	Counter := 0;
	CountFailed := 0;
END_IF

CounterOut := Counter;
CountFailedOut := CountFailed;

Camera.TubeParameters := Tube;

CASE eState OF
	E_PMLState.ePMLState_Idle: Status := 0;
	E_PMLState.ePMLState_Starting: Status := 1;
	(* put in executing to get fast answer - don't wait for execute to finish
	E_PMLState.ePMLState_Completing:
		IF Camera.Pass THEN
			Status := 2;
		ELSIF Camera.Fail THEN
			Status := 3;
		ELSIF ...
			Status := 4;
		END_IF
	*)
END_CASE

METHOD FB_init : BOOL
VAR_INPUT
	bInitRetains : BOOL; // if TRUE, the retain variables are initialized (warm start / cold start)
	bInCopyCode : BOOL;  // if TRUE, the instance afterwards gets moved into the copy code (online change)
END_VAR
IF NOT fbMessageSaved.EqualsToEventEntryEx(stOther := TC_EVENTS.SlitterEvents.ParametersSaved) THEN
	fbMessageSaved.CreateEx(TC_EVENTS.SlitterEvents.ParametersSaved, 0);
END_IF
END_METHOD

METHOD M_Aborting
M_StateComplete();

bBusy := FALSE;
bCalibration := FALSE;
Cutter.Abort();
Ejector.Abort();
Mandrel.Abort();
M_CalibrateCamera(Execute := FALSE);
Eject := FALSE;
EjectState := 0;
nCalibrationCounter := 0;

Manual.bCameraCalibrate := FALSE;
Manual.bCameraComputePeak := FALSE;
Manual.bCameraInspect := FALSE;
Manual.bCameraRawData := FALSE;
Manual.bCameraTrigger := FALSE;
Manual.bCutSample := FALSE;
Manual.bCutterDisable := FALSE;
Manual.bCutterHome := FALSE;
Manual.bCutterMoveAbs := FALSE;
Manual.bCutterReset := FALSE;
Manual.bEjectAxisEnableToggle := FALSE;
Manual.bEjectAxisFailPosition := FALSE;
Manual.bEjectAxisHomePosition := FALSE;
Manual.bEjectAxisPassPosition := FALSE;
Manual.bEjectAxisReset := FALSE;
Manual.bEjectBlowOff := FALSE;
Manual.bEjectReset := FALSE;
Manual.bEjectSamplePass := FALSE;
Manual.bEjectSampleFail := FALSE;
Manual.bEjectVacuum := FALSE;
Manual.bEjectZExtend := FALSE;
Manual.bEjectZNeutral := FALSE;
Manual.bEjectZOff := FALSE;
Manual.bEjectZRetract := FALSE;
Manual.bLowerMandrel := FALSE;
Manual.bMandrelReset := FALSE;
Manual.bMandrelSpindleRotate := FALSE;
Manual.bMandrelSpindleToggle := FALSE;
Manual.bMandrelXEnableToggle := FALSE;
Manual.bMandrelYEnableToggle := FALSE;
Manual.bMoveToCutPosition := FALSE;
Manual.bMoveToEjectPosition := FALSE;
Manual.bMoveToInspectPosition := FALSE;
Manual.bMoveToLoadPosition := FALSE;
Manual.bRaiseMandrel := FALSE;
Manual.bSaveMandrelParameters := FALSE;
Manual.bToggleMandrelVacuum := FALSE;
Manual.bVacuumAxisToggleEnable := FALSE;
Manual.bVacuumAxisMove := FALSE;
Manual.bVacuumAxisReset := FALSE;
END_METHOD

METHOD M_CalibrateCamera : INT;
VAR_INPUT
	Execute			: BOOL;
END_VAR
VAR_INST
	rTrig			: R_TRIG;
	nIndex			: INT;
	Position		: LREAL;
	debug			: INT;
	debug1			: INT;
	debug2			: INT;
END_VAR
rTrig(CLK := Execute);
IF rTrig.Q THEN
	nIndex := 10;
	Mandrel.MoveToInspectPosition(Execute := FALSE, InspectPositionX := Tube.InspectPositionX, InspectPositionY := Tube.InspectPositionY);
	Mandrel.MoveToLoadPosition(Execute := FALSE);
	Mandrel.MoveXAbs(Execute := FALSE, Position := 0);
	Mandrel.MoveYAbs(Execute := FALSE, Position := 0);
	Camera.TriggerCamera(Execute := FALSE);
	bCalibration := TRUE;
END_IF

IF NOT Execute THEN
	debug := debug + 1;
	nIndex := 0;
END_IF

CASE nIndex OF
	0: // idle state
		M_CalibrateCamera := 0;
		bCalibration := FALSE;
	10: // move to first inspection position
		IF Mandrel.MoveToInspectPosition(Execute := TRUE, InspectPositionX := Tube.InspectPositionX, InspectPositionY := Tube.InspectPositionY) = 1 THEN
			Mandrel.MoveToInspectPosition(Execute := FALSE, InspectPositionX := Tube.InspectPositionX, InspectPositionY := Tube.InspectPositionY);
			nIndex := 20;
		ELSIF Mandrel.MoveToInspectPosition(Execute := TRUE, InspectPositionX := Tube.InspectPositionX, InspectPositionY := Tube.InspectPositionY) = -1 THEN
			Mandrel.MoveToInspectPosition(Execute := FALSE, InspectPositionX := Tube.InspectPositionX, InspectPositionY := Tube.InspectPositionY);
			nIndex := 100;
		END_IF
	20: // trigger the camera
		IF Camera.TriggerCamera(Execute := TRUE) THEN
			Camera.PatternX1 := Camera.PatternMatchX;
			Camera.PatternY1 := Camera.PatternMatchY;
			Camera.TriggerCamera(Execute := FALSE);
			nIndex := 30;
		END_IF
	30: // move to second position in x
		Position := Tube.InspectPositionX + Camera.CalibrationDistance; 
		IF Mandrel.MoveXAbs(Execute := TRUE, Position := Position) = 1 THEN
			Mandrel.MoveXAbs(Execute := FALSE, Position := Position);
			nIndex := 40;
		ELSIF Mandrel.MoveXAbs(Execute := TRUE, Position := Position) = -1 THEN
			Mandrel.MoveXAbs(Execute := FALSE, Position := Position);
			nIndex := 100;
		END_IF
	40: // trigger the camera
		IF Camera.TriggerCamera(Execute := TRUE) THEN
			Camera.PatternX2 := Camera.PatternMatchX;
			Camera.PatternY2 := Camera.PatternMatchY;
			Camera.TriggerCamera(Execute := FALSE);
			nIndex := 50;
		END_IF
	45: // 
		Mandrel.MoveYAbs(Execute := FALSE, Position := 0);
		nIndex := 50;
	50: // move to the third position in y
		Position := Tube.InspectPositionY + Camera.CalibrationDistance; 
		IF Mandrel.MoveYAbs(Execute := TRUE, Position := Position) = 1 THEN
			Mandrel.MoveYAbs(Execute := FALSE, Position := Position);
			nIndex := 60;
		ELSIF Mandrel.MoveYAbs(Execute := TRUE, Position := Position) = -1 THEN
			Mandrel.MoveYAbs(Execute := FALSE, Position := Position);
			nIndex := 100;
		END_IF
	60: // trigger camera
		IF Camera.TriggerCamera(Execute := TRUE) THEN
			Camera.PatternX3 := Camera.PatternMatchX;
			Camera.PatternY3 := Camera.PatternMatchY;
			Camera.TriggerCamera(Execute := FALSE);
			nIndex := 70;
		END_IF
	70: // Calculate the pitch
		Camera.Calibrate();
		nIndex := 80; 
	80: // return to load position	
		IF Mandrel.MoveToLoadPosition(Execute := TRUE) <> 0 THEN
			Mandrel.MoveToLoadPosition(Execute := FALSE);
			nIndex := 90;
		END_IF
	90: // done state
		M_CalibrateCamera := 1;
	 
	100: // error state
		M_CalibrateCamera := -1;
	
END_CASE
END_METHOD

METHOD M_Clearing
CASE eMode OF
	E_PMLProtectedUnitMode.ePMLProtUnitMode_Manual: M_ClearingManual();
	
	E_PMLProtectedUnitMode.ePMLProtUnitMode_Production: M_ClearingProduction();
END_CASE
END_METHOD

METHOD M_ClearingManual : BOOL
VAR_INPUT
END_VAR
M_StateComplete();
//M_ClearingManual := TRUE;
END_METHOD

METHOD M_ClearingProduction : BOOL
VAR_INPUT
END_VAR
CASE nState OF
	0:	// reset the variables
		Mandrel.Clear(Execute := FALSE);
		Cutter.Clear(Execute := FALSE);
		Ejector.Reset(Execute := FALSE);
		nState := 10;
	10: // reset the cutter
		IF Cutter.Clear(Execute := TRUE) = 1 THEN
			Cutter.Clear(Execute := FALSE);
			nState := 20;
		END_IF	
	20: // reset the ejector
		IF Ejector.Reset(Execute := TRUE) = 1 THEN
			Ejector.Reset(Execute := FALSE);
			nState := 30;		END_IF

	30: // reset the different objects
		IF Mandrel.Clear(Execute := TRUE) = 1 THEN
			Mandrel.Clear(Execute := FALSE);
			nState := 40;
		END_IF
	40:	// done state
		M_StateComplete();
END_CASE
END_METHOD


METHOD M_Complete
END_METHOD

METHOD M_Completing

VAR
	EjectSample: INT;
END_VAR
IF eMode = E_PMLProtectedUnitMode.ePMLProtUnitMode_Production THEN
	CASE EjectState OF
		0: // wait for eject command
			M_StateComplete();
		10: // execute the eject pass sequence
			EjectSample := Ejector.EjectSamplePass(Execute := TRUE);
			IF EjectSample = 1 THEN
				Eject := FALSE;
				Ejector.EjectSamplePass(Execute := FALSE);
				EjectState := 0;
			ELSIF EjectSample = -1 THEN
				Eject := FALSE;
				EjectState := 0;
				Ejector.EjectSamplePass(Execute := FALSE);
			END_IF
		20: // execute the eject fail sequence
			EjectSample := Ejector.EjectSampleFail(Execute := TRUE);
			IF EjectSample = 1 THEN
				Eject := FALSE;
				Ejector.EjectSampleFail(Execute := FALSE);
				EjectState := 0;
			ELSIF EjectSample = -1 THEN
				Eject := FALSE;
				EjectState := 0;
				Ejector.EjectSampleFail(Execute := FALSE);
			END_IF
	END_CASE
ELSE
	M_StateComplete();
END_IF
END_METHOD

METHOD M_Execute
VAR_INST
	Result					: INT;
END_VAR
VAR
	CutPositionY 			: LREAL;
	VelocityY 				: LREAL;
	MoveToCutPosition 		: INT;
	MoveToInspectPosition 	: INT;
	MoveToEjectPosition 	: INT;
	MoveToLoadPosition 		: INT;
	CutSample				: INT;
	EjectSample 			: INT;

	CameraIndex 			: INT;
	FileName				: STRING;
	FilePath				: STRING;
	RotateDistance			: LREAL;
END_VAR
VAR_INST
	StrResult				: STRING(255);
	SampleLowered			: BOOL;
	LiftTon					: TON := (PT := T#500MS);
	VacuumSensorTON			: TON := (PT := T#2S);
	hFile					: UINT;
	AttemptCounter			: INT;
	Pass					: BOOL;
	Message					: STRING(255);
END_VAR
Eject := FALSE;
fbLocalSystemTime(
	sNetId := '',
	bEnable := TRUE,
	dwCycle := 1);

IF eMode = E_PMLProtectedUnitMode.ePMLProtUnitMode_Production THEN
	CASE nState OF
		0: // do we need to write to the camera?
			AttemptCounter := 0;
			bDecrementSpindle:= FALSE;
			bIncrementSpindle:= FALSE;
			bInspect:= FALSE;
			bInspectComplete:= FALSE;

			SampleLowered := FALSE;
			VacuumSensorTON(IN := FALSE);
			Result := Camera.SelectCameraProgram(Execute := TRUE);
			IF Result = 1 THEN
				Camera.SelectCameraProgram(Execute := FALSE);
				nState := 5;
			ELSIF Result = -1 THEN
				Camera.SelectCameraProgram(Execute := FALSE);
				Message := 'Camera failed to read/write to modbus.';
				nState := 666;
			END_IF
		5: // move the vacuum axis to the correct location
			IF Mandrel.MoveToVacPosition(Execute := TRUE) THEN
				Mandrel.MoveToVacPosition(Execute := FALSE);
				nState := 10;
			END_IF
		10: // turn on mandrel vacuum and move to cut position
			Mandrel.MandrelVacuum := TRUE;
			IF Mandrel.LowerSample() = 1 THEN
				SampleLowered := TRUE;
				nState := 11;
			END_IF
		11: // wait for vacuum sensor to detect the tube
			VacuumSensorTON(IN := TRUE);
			IF Mandrel.VacuumSensor > Tube.VacuumThreshold THEN
				nState := 15;
				VacuumSensorTON(IN := FALSE);
			END_IF
			IF VacuumSensorTON.Q THEN
				Mandrel.MandrelVacuum := FALSE;
				nState := 110;
				VacuumSensorTON(IN := FALSE);
			END_IF
		15: // move to cut position
			MoveToCutPosition := Mandrel.MoveToCutPosition(Execute := TRUE, CutPositionX := Tube.CutPositionX, CutPositionY := Tube.CutPositionY);
			IF MoveToCutPosition = 1 AND SampleLowered THEN
				Mandrel.MoveToCutPosition(Execute := FALSE, CutPositionX := Tube.CutPositionX, CutPositionY := Tube.CutPositionY);
				nState := 20;
				SampleLowered := FALSE;
			ELSIF MoveToCutPosition = -1 THEN
				Mandrel.MoveToCutPosition(Execute := FALSE, CutPositionX := Tube.CutPositionX, CutPositionY := Tube.CutPositionY);
				nState := 666;
				Message := 'Mandrel failed to move.';
				SampleLowered := FALSE;
			END_IF
		20: // make a cut unless we are just inspecting
			IF Inspect THEN
				nState := 30;
			ELSE
				CutSample := Cutter.CutSample(Execute := TRUE);
				IF CutSample = 1 THEN
					Cutter.CutSample(Execute := FALSE);
					nState := 30;
				ELSIF CutSample = -1 THEN
					Cutter.CutSample(Execute := FALSE);
					nState := 666;
				END_IF
			END_IF
		30: // raise sample
			// move to inspect position
			Mandrel.LiftSample();
			MoveToInspectPosition := Mandrel.MoveToInspectPosition(Execute := TRUE, InspectPositionX := Tube.InspectPositionX, InspectPositionY := Tube.InspectPositionY);
			IF MoveToInspectPosition = 1 THEN
				Mandrel.MoveToInspectPosition(Execute := FALSE, InspectPositionX := Tube.InspectPositionX, InspectPositionY := Tube.InspectPositionY);
				nState := 35;
			ELSIF MoveToInspectPosition = -1 THEN
				Mandrel.MoveToInspectPosition(Execute := FALSE, InspectPositionX := Tube.InspectPositionX, InspectPositionY := Tube.InspectPositionY);
				nState := 666;
			END_IF
		35: // add 500 ms delay for lifter
			LiftTON.IN := TRUE;
			IF LiftTON.Q THEN
				LiftTON.IN := FALSE;
				IF Inspect THEN
					nState := 36;
				ELSE
					nState := 40;
				END_IF
			END_IF
			LiftTON();
		36: // Inspect under manual control
			Result := Camera.Inspect(Execute := TRUE);
			IF Result = 1 THEN
				nState := 37;
				Camera.Inspect(Execute := FALSE);
				IF Camera.Pass THEN
					Status := 2;
				ELSE
					Status := 3;
				END_IF
			ELSIF Result = -1 THEN
				Status := 4;
				nState := 37;
			END_IF
			//nState := 37;
		37: // wait for command
			IF bDecrementSpindle THEN
				bDecrementSpindle := FALSE;
				nState := 39;
			ELSIF bIncrementSpindle THEN
				bIncrementSpindle := FALSE;
				nState := 38;
			ELSIF bInspect THEN
				bInspect := FALSE;
				nState := 36;
			ELSIF bInspectComplete THEN
				bInspectComplete := FALSE;
				nState := 70;
			END_IF
		38: // increment spindle
			IF Mandrel.RotateSpindle(Execute := TRUE, Distance := Mandrel.SpindleIncrement ) <> 0 THEN
				Mandrel.RotateSpindle(Execute := FALSE, Distance := Mandrel.SpindleIncrement);
				nState := 37;
			END_IF
		39: // decrement spindle
			IF Mandrel.RotateSpindle(Execute := TRUE, Distance := -1 * Mandrel.SpindleIncrement) <> 0 THEN
				Mandrel.RotateSpindle(Execute := FALSE, Distance := -1 * Mandrel.SpindleIncrement);
				nState := 37;
			END_IF
			
		40: // inspect
			Result := Camera.Inspect(Execute := TRUE);
			IF Result = 1 THEN
				Camera.Inspect(Execute := FALSE);
				IF Camera.Pass THEN
					Mandrel.MandrelVacuum := FALSE;
					IF Manual.bCalibrateMandrel THEN
						CalibrationArrayX[nCalibrationCounter] := Camera.DeltaXmmWithOffset;
						CalibrationArrayY[nCalibrationCounter] := Camera.DeltaYmmWithOffset;
						nCalibrationCounter := nCalibrationCounter + 1;
						IF nCalibrationCounter > CalMax THEN
							MandrelCalibration();
							Manual.bCalibrateMandrel := FALSE;
							nCalibrationCounter := 0;
						END_IF
					END_IF
					Pass := TRUE;
					nState := 50;	// passed -> go to eject pass station
					Status := 2;
				ELSE
					Mandrel.MandrelVacuum := FALSE;
					Pass := FALSE;
					nState := 50;	// failed -> go to eject fail station
					Status := 3;
				END_IF
			ELSIF Result = -1 THEN	// couldn't find the pattern; need to advance the counter and retry
				AttemptCounter := AttemptCounter + 1;
				Camera.Inspect(Execute := FALSE);
				IF AttemptCounter > 3 THEN	// error
					nState := 70;			// error out
					Status := 4;
				ELSE						// advance the motor a bit and retry
					nState := 45;
				END_IF
			END_IF
		45: // advance the tube a bit and then go and retry the process
			Result := Mandrel.MoveXRel(Execute := TRUE, Distance := 1);
			IF Result = 1 THEN
				Mandrel.MoveXRel(Execute := FALSE, Distance := 1);
				nState := 35;
			END_IF
			
		50: // move to eject position		
			MoveToEjectPosition := Mandrel.MoveToEjectPosition(Execute := TRUE, EjectPositionX := Tube.EjectPositionX, EjectPositionY := Tube.EjectPositionY);
			IF MoveToEjectPosition = 1 THEN
				Mandrel.MoveToEjectPosition(Execute := FALSE, EjectPositionX := Tube.EjectPositionX, EjectPositionY := Tube.EjectPositionY);
				nState := 60;
			ELSIF MoveToEjectPosition = -1 THEN
				Mandrel.MoveToEjectPosition(Execute := FALSE, EjectPositionX := Tube.EjectPositionX, EjectPositionY := Tube.EjectPositionY);
				nState := 666;
			END_IF
		60: // do the eject sequence 
			Eject := TRUE;		
			// wait for the system to retract
			IF Ejector.IsEjectZExtend THEN
				nState := 65;
			END_IF
		65: // wait for ejector actuator to be clear to retract the mandrel
			IF Ejector.IsEjectZRetract THEN
				nState := 70;
			END_IF 
		70: // move to load position
			Mandrel.MandrelVacuum := FALSE;

			IF Mandrel.LowerSample() = 1 THEN
				SampleLowered := TRUE;
			END_IF
			IF Manual.bCalibrateMandrel THEN
				IF Mandrel.SpindleOffset >= 0 THEN
					RotateDistance := (360.0 / (INT_TO_LREAL(CalMax)+1.0)) - Mandrel.SpindleOffset;
				ELSE
					RotateDistance := -1 * ( (360.0 / (INT_TO_LREAL(CalMax)+1.0)) + Mandrel.SpindleOffset);
				END_IF
				IF Mandrel.RotateSpindle(Execute := TRUE, Distance := RotateDistance) <> 0 THEN
					Mandrel.RotateSpindle(Execute := FALSE, Distance := RotateDistance);
					nState := 75;
				END_IF
			ELSE
				nState := 75;			
			END_IF
		75: // move to load position cont'd
			IF Mandrel.LowerSample() = 1 THEN
				SampleLowered := TRUE;
			END_IF

			MoveToLoadPosition := Mandrel.MoveToLoadPosition(Execute := TRUE);
			IF MoveToLoadPosition = 1 AND SampleLowered THEN
				Mandrel.MoveToLoadPosition(Execute := FALSE);
				SampleLowered := FALSE;
				nState := 80;
			ELSIF MoveToLoadPosition = -1 THEN
				SampleLowered := FALSE;
				Mandrel.MoveToLoadPosition(Execute := FALSE);
				nState := 666;
			END_IF
		80: // check if vacuum is off
			IF Mandrel.VacuumSensor < Tube.VacuumThreshold THEN
				nState := 90;
				Mandrel.MandrelVacuum := FALSE;
			END_IF
		90:	// increment counters state
			IF NOT Inspect THEN			
				Counter := Counter + 1;
				IF NOT Camera.Pass THEN
					CountFailed := CountFailed + 1;
				END_IF
				nState := 100;
			ELSE
				nState := 110;
			END_IF			
		100: // save to file
			FileName := CONCAT(ULINT_TO_STRING(Batch), '.txt');
			FilePath := CONCAT('D:\',FileName);
			fbFileOpen(
				sNetId := '',
				sPathName := FilePath,
				nMode := FOPEN_MODEAPPEND,
				ePath := E_OpenPath.PATH_GENERIC,
				hFile => hFile,
				bExecute := TRUE);
			IF NOT fbFileOpen.bBusy THEN
				fbFileOpen(
					sNetId := '',
					sPathName := FilePath,
					nMode := FOPEN_MODEAPPEND,
					ePath := E_OpenPath.PATH_GENERIC,
					bExecute := FALSE);
				nState := 101;
			END_IF
			IF fbFileOpen.bError THEN
				fbFileOpen(
					sNetId := '',
					sPathName := FilePath,
					nMode := FOPEN_MODEAPPEND,
					ePath := E_OpenPath.PATH_GENERIC,
					bExecute := FALSE);
				nState := 102;				
			END_IF
		101: // write data to file	
			StrResult := '';		
			StrResult := CONCAT(ULINT_TO_STRING(Batch), ', ');
			StrResult := CONCAT(StrResult, UINT_TO_STRING(Counter));
			StrResult := CONCAT(StrResult, ', ');
			// add the system time
			IF fbLocalSystemTime.bValid THEN
				StrResult := CONCAT(StrResult, SYSTEMTIME_TO_STRING(fbLocalSystemTime.systemTime));
				StrResult := CONCAT(StrResult, ', ');
			END_IF
			IF Camera.Pass THEN
				StrResult := CONCAT(StrResult, 'PASS, ');
			ELSIF Camera.Fail THEN
				StrResult := CONCAT(StrResult, 'FAIL, ');
			ELSIF Camera.NoDetect THEN
				StrResult := CONCAT(StrResult, 'NO DETECT, ');
			END_IF
			IF NOT Camera.NoDetect THEN
				StrResult := CONCAT(StrResult, 'x := ');
				StrResult := CONCAT(StrResult, REAL_TO_STRING(Camera.DeltaXmmWithOffset));
				StrResult := CONCAT(StrResult, ', y := ');
				StrResult := CONCAT(StrResult, REAL_TO_STRING(Camera.DeltaYmmWithOffset));
				StrResult := CONCAT(StrResult, ', length := ');
				StrResult := CONCAT(StrResult, REAL_TO_STRING(Camera.CutLengthWithOffset));
			ELSE
				StrResult := CONCAT(StrResult, 'x := not detected');
				StrResult := CONCAT(StrResult, ', y := not detected');
				StrResult := CONCAT(StrResult, ', length := not detected');			
			END_IF
			StrResult := CONCAT(StrResult, '$r$n');
			fbFileWrite(
				sNetId := '',
				hFile := hFile,
				pWriteBuff := ADR(StrResult),
				cbWriteLen := INT_TO_UINT(LEN(StrResult)),
				bExecute := TRUE
			);
			IF NOT fbFileWrite.bBusy THEN
				nState := 102;
				fbFileWrite(bExecute := FALSE);
			END_IF
			IF fbFileWrite.bError THEN
				nState := 102;
				fbFileWrite(bExecute := FALSE);
			END_IF
		102: // file close
			fbFileClose(
				sNetId := '',
				hFile := hFile,
				bExecute := TRUE);
			IF NOT fbFileClose.bBusy THEN
				fbFileClose(bExecute := FALSE);
				nState := 110;
			END_IF
			IF fbFileClose.bError THEN
				fbFileClose(bExecute := FALSE);
				nState := 110;
			END_IF
		110: // done state
			M_StateComplete();
	END_CASE
	
	CASE EjectState OF
		0: // wait for eject command
			Ejector.EjectSamplePass(Execute := FALSE);
			Ejector.EjectSampleFail(Execute := FALSE);
			IF Eject AND Pass THEN
				EjectState := 10;
			ELSIF Eject AND NOT Pass THEN
				EjectState := 20;
			END_IF
		10: // execute the eject pass sequence
			EjectSample := Ejector.EjectSamplePass(Execute := TRUE);
			IF EjectSample = 1 THEN
				Eject := FALSE;
				Ejector.EjectSamplePass(Execute := FALSE);
				EjectState := 0;
			ELSIF EjectSample = -1 THEN
				Eject := FALSE;
				EjectState := 0;
				Ejector.EjectSamplePass(Execute := FALSE);
			END_IF
		20: // execute the eject fail sequence
			EjectSample := Ejector.EjectSampleFail(Execute := TRUE);
			IF EjectSample = 1 THEN
				Eject := FALSE;
				Ejector.EjectSampleFail(Execute := FALSE);
				EjectState := 0;
			ELSIF EjectSample = -1 THEN
				Eject := FALSE;
				EjectState := 0;
				Ejector.EjectSampleFail(Execute := FALSE);
			END_IF

	END_CASE
ELSIF eMode = E_PMLProtectedUnitMode.ePMLProtUnitMode_Manual THEN
	M_Manual();
END_IF
END_METHOD


METHOD M_Held
END_METHOD


METHOD M_Holding
END_METHOD


METHOD M_Idle
END_METHOD

METHOD M_Manual : BOOL
VAR_INPUT
END_VAR
VAR_INST
	Operational	: BOOL;
	Result		: INT;
	TON			: TON := (PT := T#5S);
	x			: INT;
END_VAR

IF Manual.bCameraCalibrate THEN
	bBusy := TRUE;
	IF M_CalibrateCamera(Execute := TRUE) <> 0 THEN
		M_CalibrateCamera(Execute := FALSE);
		bBusy := FALSE;
		Manual.bCameraCalibrate := FALSE;
	END_IF
END_IF

IF Manual.bCameraComputePeak THEN
	bBusy := TRUE;
	IF Camera.Compute(Execute := TRUE) = 1 THEN
		bBusy := FALSE;
		Camera.Compute(Execute := FALSE);
		Manual.bCameraComputePeak := FALSE;
	END_IF
END_IF

IF Manual.bCameraInspect THEN
	bBusy := TRUE;
	IF Camera.Inspect(Execute := TRUE) = 1 THEN
		Camera.Inspect(Execute := FALSE);
		Manual.bCameraInspect := FALSE;
		bBusy := FALSE;
	END_IF
END_IF	

IF Manual.bCameraRawData THEN
	bBusy := TRUE;
	IF Camera.GetCameraData() <> 0 THEN
		bBusy := FALSE;
		Manual.bCameraRawData := FALSE;
	END_IF
END_IF

IF Manual.bCameraSelectTube THEN
	bBusy := TRUE;
	Result := Camera.SelectCameraProgram(Execute := TRUE);
	IF Result = 1 THEN
		bBusy := FALSE;
		Manual.bCameraSelectTube := FALSE;
		Camera.SelectCameraProgram(Execute := FALSE);
	ELSIF Result = -1 THEN
		bBusy := FALSE;
		Manual.bCameraSelectTube := FALSE;
		Camera.SelectCameraProgram(Execute := FALSE);
		x := x + 1;
	END_IF
END_IF

IF Manual.bCameraTrigger THEN
	bBusy := TRUE;
	IF Camera.TriggerCamera(Execute := TRUE) THEN
		Camera.TriggerCamera(Execute := FALSE);
		bBusy := FALSE;
		Manual.bCameraTrigger := FALSE;
	END_IF
END_IF

IF Manual.bCutSample THEN
	bBusy := TRUE;
	IF Cutter.CutSample(Execute := TRUE) <> 0 THEN
		Cutter.CutSample(Execute := FALSE);
		Manual.bCutSample := FALSE;
		bBusy := FALSE;
	END_IF
END_IF

IF Manual.bCutterDisable THEN
	IF NOT bBusy THEN
		Operational := Cutter.IsEnabled;
		TON(IN := TRUE);
	END_IF
	bBusy := TRUE;
	IF Operational THEN
		IF Cutter.Disable() THEN
			TON(IN := FALSE);
			bBusy := FALSE;
			Manual.bCutterDisable := FALSE;
		END_IF
	ELSE
		IF Cutter.Enable() OR TON.q	THEN
			bBusy := FALSE;
			TON(IN := FALSE);
			Manual.bCutterDisable := FALSE;
		END_IF
	END_IF
	TON();
END_IF

IF Manual.bCutterHome THEN
	bBusy := TRUE;
	IF Cutter.Home(Execute := TRUE) <> 0 THEN
		bBusy := FALSE;
		Cutter.Home(Execute := FALSE);
		Manual.bCutterHome := FALSE;
	END_IF
END_IF

IF Manual.bCutterMoveAbs THEN
	bBusy := FALSE;
	IF Cutter.MoveAbs(Execute := TRUE) <> 0 THEN
		bBusy := FALSE;
		Cutter.MoveAbs(Execute := FALSE);
		Manual.bCutterMoveAbs := FALSE;
	END_IF
END_IF

IF Manual.bCutterReset THEN
	bBusy := TRUE;
	IF Cutter.Reset(Execute := TRUE) <> 0 THEN
		bBusy := FALSE;
		Manual.bCutterReset := FALSE;
		Cutter.Reset(Execute := FALSE);
	END_IF
END_IF

IF Manual.bEjectBlowOff THEN
	Ejector.BlowOff := NOT Ejector.BlowOff;
	Manual.bEjectBlowOff := FALSE;
END_IF

IF Manual.bEjectSamplePass THEN
	bBusy := TRUE;
	IF Ejector.EjectSamplePass(Execute := TRUE) = 1 THEN
		Ejector.EjectSamplePass(Execute := FALSE);
		Manual.bEjectSamplePass := FALSE;
		bBusy := FALSE;
	END_IF
END_IF

IF Manual.bEjectSampleFail THEN
	bBusy := TRUE;
	IF Ejector.EjectSampleFail(Execute := TRUE) = 1 THEN
		Ejector.EjectSampleFail(Execute := FALSE);
		Manual.bEjectSampleFail := FALSE;
		bBusy := FALSE;
	END_IF
END_IF

IF Manual.bEjectVacuum THEN
	Ejector.PickUpVacuum := NOT Ejector.PickUpVacuum;
	Manual.bEjectVacuum := FALSE;
END_IF
(*
	bEjectAxisPassPosition	: BOOL;
	bEjectAxisHomePosition	: BOOL;
	bEjectAxisFailPosition	: BOOL;
	bEjectAxisEnable		: BOOL;
	bEjectAxisDisabe		: BOOL;
	bEjectAxisReset			: BOOL;
	bEjectSamplePass		: BOOL;
	bEjectSampleFail		: BOOL;
*)
IF Manual.bEjectAxisEnableToggle THEN
	IF NOT bBusy THEN
		Operational := Ejector.axis.IsEnabled;
	END_IF
	bBusy := TRUE;
	IF Operational THEN
		IF Ejector.axis.Disable() THEN
			bBusy := FALSE;
			Manual.bEjectAxisEnableToggle := FALSE;
		END_IF
	ELSE
		IF Ejector.axis.Enable() THEN
			bBusy := FALSE;
			Manual.bEjectAxisEnableToggle := FALSE;
		END_IF		
	END_IF
END_IF

IF Manual.bEjectAxisFailPosition THEN
	bBusy := TRUE;
	IF Ejector.axis.AbsMove(Execute := TRUE, 
		Position := Ejector.EjectAxisFailPosition, 
		Velocity := Ejector.EjectAxisVelocity) THEN
			Ejector.axis.AbsMove(Execute := FALSE, Position := Ejector.EjectAxisFailPosition, Velocity := Ejector.EjectAxisVelocity);	
			bBusy := FALSE;
			Manual.bEjectAxisFailPosition := FALSE;
	END_IF
END_IF

IF Manual.bEjectAxisHomePosition THEN
	bBusy := TRUE;
	IF Ejector.axis.AbsMove(Execute := TRUE, 
		Position := Ejector.EjectAxisHomePosition, 
		Velocity := Ejector.EjectAxisVelocity) THEN
			Ejector.axis.AbsMove(Execute := FALSE, Position := Ejector.EjectAxisHomePosition, Velocity := Ejector.EjectAxisVelocity);
			bBusy := FALSE;
			Manual.bEjectAxisHomePosition := FALSE;
	END_IF
END_IF

IF Manual.bEjectAxisPassPosition THEN
	bBusy := TRUE;
	IF Ejector.axis.AbsMove(Execute := TRUE, 
		Position := Ejector.EjectAxisPassPosition, 
		Velocity := Ejector.EjectAxisVelocity) THEN
			Ejector.axis.AbsMove(Execute := FALSE, Position := Ejector.EjectAxisPassPosition, Velocity := Ejector.EjectAxisVelocity);
			bBusy := FALSE;
			Manual.bEjectAxisPassPosition := FALSE;
	END_IF
END_IF

IF Manual.bEjectAxisReset THEN
	bBusy := TRUE;
	IF Ejector.axis.Reset(Execute := TRUE) THEN
		Ejector.axis.Reset(Execute := FALSE);
		bBusy := FALSE;
		Manual.bEjectAxisReset := FALSE;
	END_IF
END_IF

IF Manual.bEjectReset THEN
	bBusy := TRUE;
	IF Ejector.Reset(TRUE) = 1 THEN
		Ejector.Reset(FALSE);
		bBusy := FALSE;
		Manual.bEjectReset := FALSE;
	END_IF
END_IF

IF Manual.bEjectZExtend THEN
	bBusy := TRUE;
	IF Ejector.zSlide.Extend() = 1 THEN
		bBusy := FALSE;
		Manual.bEjectZExtend := FALSE;
	END_IF
END_IF

IF Manual.bEjectZNeutral THEN
	bBusy := TRUE;
	IF Ejector.zSlide.Neutral() THEN
		bBusy := FALSE;
		Manual.bEjectZNeutral := FALSE;
	END_IF
END_IF

IF Manual.bEjectZRetract THEN
	bBusy := TRUE;
	IF Ejector.zSlide.Retract() = 1 THEN
		bBusy := FALSE;
		Manual.bEjectZRetract := FALSE;
	END_IF
END_IF

IF Manual.bLowerMandrel THEN
	bBusy := TRUE;
	IF Mandrel.LowerSample() = 1 THEN
		bBusy := FALSE;
		Manual.bLowerMandrel := FALSE;
	END_IF
END_IF

IF Manual.bMandrelSpindleRotate THEN
	bBusy := TRUE;
	IF Mandrel.RotateSpindle(Execute := TRUE, Distance := Mandrel.SpindleIncrement) <> 0 THEN
		bBusy := FALSE;
		Mandrel.RotateSpindle(Execute := FALSE, Distance := Mandrel.SpindleIncrement);
		Manual.bMandrelSpindleRotate := FALSE;
	END_IF
END_IF

IF Manual.bMandrelSpindleToggle THEN
	IF NOT bBusy THEN
		Operational := Mandrel.OperationalSpindle;
	END_IF
	bBusy := TRUE;
	IF Operational THEN
		IF Mandrel.DisableSpindle() THEN
			bBusy := FALSE;
			Manual.bMandrelSpindleToggle := FALSE;
		END_IF
	ELSE
		IF Mandrel.EnableSpindle() THEN
			bBusy := FALSE;
			Manual.bMandrelSpindleToggle := FALSE;
		END_IF
	END_IF
END_IF

IF Manual.bMandrelXEnableToggle THEN
	IF NOT bBusy THEN
		Operational := Mandrel.OperationalX;
	END_IF
	bBusy := TRUE;
	IF Operational THEN
		IF Mandrel.DisableX() THEN
			bBusy := FALSE;
			Manual.bMandrelXEnableToggle := FALSE;
		END_IF
	ELSE
		IF Mandrel.EnableX() THEN
			bBusy := FALSE;
			Manual.bMandrelXEnableToggle := FALSE;
		END_IF
	END_IF	
END_IF

IF Manual.bMandrelYEnableToggle THEN
	IF NOT bBusy THEN
		Operational := Mandrel.OperationalY;
	END_IF
	bBusy := TRUE;
	IF Operational THEN
		IF Mandrel.DisableY() THEN
			bBusy := FALSE;
			Manual.bMandrelYEnableToggle := FALSE;
		END_IF
	ELSE
		IF Mandrel.EnableY() THEN
			bBusy := FALSE;
			Manual.bMandrelYEnableToggle := FALSE;
		END_IF
	END_IF		
END_IF

IF Manual.bMandrelReset THEN
	bBusy := TRUE;
	IF Mandrel.Reset(Execute := TRUE) = 1 THEN
		Mandrel.Reset(Execute := FALSE);
		bBusy := FALSE;
		Manual.bMandrelReset := FALSE;
	END_IF
END_IF

IF Manual.bMoveToCutPosition THEN
	bBusy := TRUE;
	IF Mandrel.MoveToCutPosition(Execute := TRUE, CutPositionX := TubeHmi.CutPositionX, CutPositionY := TubeHmi.CutPositionY ) = 1 THEN
		Mandrel.MoveToCutPosition(Execute := FALSE, CutPositionX := TubeHmi.CutPositionX, CutPositionY := TubeHmi.CutPositionY);
		Manual.bMoveToCutPosition := FALSE;
		bBusy := FALSE;
	END_IF
END_IF

IF Manual.bMoveToEjectPosition THEN
	bBusy := TRUE;
	IF Mandrel.MoveToEjectPosition(Execute := TRUE, EjectPositionX := TubeHmi.EjectPositionX, EjectPositionY := TubeHmi.EjectPositionY) = 1 THEN
		Mandrel.MoveToEjectPosition(Execute := FALSE, EjectPositionX := TubeHmi.EjectPositionX, EjectPositionY := TubeHmi.EjectPositionY);
		Manual.bMoveToEjectPosition := FALSE;
		bBusy := FALSE;
	END_IF
END_IF

IF Manual.bMoveToInspectPosition THEN
	bBusy := TRUE;
	IF Mandrel.MoveToInspectPosition(Execute := TRUE, InspectPositionX := TubeHmi.InspectPositionX, InspectPositionY := TubeHmi.InspectPositionY) = 1 THEN
		Mandrel.MoveToInspectPosition(Execute := FALSE, InspectPositionX := TubeHmi.InspectPositionX, InspectPositionY := TubeHmi.InspectPositionY);
		Manual.bMoveToInspectPosition := FALSE;
		bBusy := FALSE;
	END_IF
END_IF

IF Manual.bMoveToLoadPosition THEN
	bBusy := TRUE;
	IF Mandrel.MoveToLoadPosition(Execute := TRUE) = 1 THEN
		Mandrel.MoveToLoadPosition(Execute := FALSE);
		Manual.bMoveToLoadPosition := FALSE;
		bBusy := FALSE;
	END_IF
END_IF

IF Manual.bRaiseMandrel THEN
	bBusy := TRUE;
	IF Mandrel.LiftSample() = 1 THEN
		bBusy := FALSE;
		Manual.bRaiseMandrel := FALSE;
	END_IF
END_IF

IF Manual.bToggleMandrelVacuum THEN
	Mandrel.MandrelVacuum := NOT Mandrel.MandrelVacuum;
	Manual.bToggleMandrelVacuum := FALSE;
END_IF


IF Manual.bVacuumAxisMove THEN
	bBusy := TRUE;
	IF Mandrel.VacAxis.AbsMove(Execute := TRUE, Position := TubeHmi.VacPosition, Velocity := Mandrel.VacuumVelocity) THEN
		Mandrel.VacAxis.AbsMove(Execute := FALSE, Position := 0, Velocity := 0);
		bBusy := FALSE;
		Manual.bVacuumAxisMove := FALSE;
	END_IF
END_IF

IF Manual.bVacuumAxisReset THEN
	bBusy := TRUE;
	IF Mandrel.VacAxis.Reset(Execute := TRUE) THEN
		Mandrel.VacAxis.Reset(Execute := FALSE);
		bBusy := FALSE;
		Manual.bVacuumAxisReset := FALSE;
	END_IF
END_IF

IF Manual.bVacuumAxisToggleEnable THEN
	IF NOT bBusy THEN
		Operational := Mandrel.VacAxis.IsEnabled;
	END_IF
	bBusy := TRUE;
	IF Operational THEN
		IF Mandrel.VacAxis.Disable() THEN
			bBusy := FALSE;
			Manual.bVacuumAxisToggleEnable := FALSE;
		END_IF
	ELSE
		IF Mandrel.VacAxis.Enable() THEN
			bBusy := FALSE;
			Manual.bVacuumAxisToggleEnable := FALSE;
		END_IF
	END_IF
END_IF
END_METHOD

METHOD M_Production : BOOL
VAR_INPUT
END_VAR
END_METHOD

METHOD M_Resetting
M_StateComplete();
END_METHOD

METHOD M_Starting
Mandrel.MoveToCutPosition(Execute := FALSE, CutPositionX := Tube.CutPositionX, CutPositionY := Tube.CutPositionY);
Cutter.CutSample(Execute := FALSE);
Mandrel.MoveToInspectPosition(Execute := FALSE, InspectPositionX := Tube.InspectPositionX, InspectPositionY := Tube.InspectPositionY);
Camera.Inspect(Execute := FALSE);
Mandrel.MoveToEjectPosition(Execute := FALSE, EjectPositionX := Tube.EjectPositionX, EjectPositionY := Tube.EjectPositionY);
Mandrel.MoveToLoadPosition(Execute := FALSE);
Camera.SelectCameraProgram(Execute := FALSE);
//Mandrel.MoveToVacPosition(Execute := FALSE);
fbFileOpen(bExecute := FALSE);
fbFileWrite(bExecute := FALSE);
fbFileClose(bExecute := FALSE);

IF Mandrel.LowerSample() = 1 THEN
	M_StateComplete();
END_IF
END_METHOD


METHOD M_Stopped
END_METHOD


METHOD M_Stopping
END_METHOD


METHOD M_Suspended
END_METHOD


METHOD M_Suspending
END_METHOD


METHOD M_Undefined
END_METHOD


METHOD M_Unholding
END_METHOD


METHOD M_Unsuspending
END_METHOD

METHOD MandrelCalibration : BOOL
VAR_INPUT
END_VAR

VAR
	i: INT;
	SumX: LREAL;
	SumY: LREAL;
END_VAR
SumX := 0;
SumY := 0;
FOR i:= 0 TO CalMax DO
	SumX := CalibrationArrayX[i] + SumX;
	SumY := CalibrationArrayY[i] + SumY;
END_FOR
AverageX := SumX / 10.0;
AverageY := SumY / 10.0;

Tube.CutPositionX := Tube.CutPositionX - AverageX;
Tube.CutPositionY := Tube.CutPositionY - AverageY;
END_METHOD

PROPERTY MandrelVacuum : BOOL
GET
MandrelVacuum := Mandrel.MandrelVacuum;
END_GET
SET
Mandrel.MandrelVacuum := MandrelVacuum;
END_SET
END_PROPERTY

METHOD ReadParameters : BOOL
VAR_INPUT
	Execute	: BOOL;
END_VAR
VAR_INST
	nReadIndex	: INT;
	rTrig		: R_TRIG;
END_VAR
ReadParameters := FALSE;
rTrig(CLK := Execute);
IF rTrig.Q THEN
	nReadIndex := 5;
END_IF

IF NOT Execute THEN
	nReadIndex := 0;
END_IF

CASE nReadIndex OF
	5: // read the info from the config file for the camera
		fbXmlSrvRead.sXPath := '/Configuration/Camera';
		fbXmlSrvRead.pSymAddr := ADR(CameraParameters);
		fbXmlSrvRead.cbSymSize := SIZEOF(CameraParameters);
		fbXmlSrvRead.bExecute := TRUE;
		nReadIndex := 10;
	10: // wait for the info to load
		IF NOT fbXmlSrvRead.bBusy THEN
			fbXmlSrvRead.bExecute := FALSE;
			Camera.Parameters := CameraParameters;
			nReadIndex := 20;
		END_IF
	20: // read the info from the config file for the cutter
		fbXmlSrvRead.sXPath := '/Configuration/Cutter';
		fbXmlSrvRead.pSymAddr := ADR(CutterParameters);
		fbXmlSrvRead.cbSymSize := SIZEOF(CutterParameters);
		fbXmlSrvRead.bExecute := TRUE;
		nReadIndex := 30;
	30: // wait to complete
		IF NOT fbXmlSrvRead.bBusy THEN
			fbXmlSrvRead.bExecute := FALSE;
			Cutter.Parameters := CutterParameters;
			nReadIndex := 40;
		END_IF
	40: // read the ejector parameters
		fbXmlSrvRead.sXPath := '/Configuration/Ejector';
		fbXmlSrvRead.pSymAddr := ADR(EjectorParameters);
		fbXmlSrvRead.cbSymSize := SIZEOF(EjectorParameters);
		fbXmlSrvRead.bExecute := TRUE;
		nReadIndex := 50;
	50: // wait
		IF NOT fbXmlSrvRead.bBusy THEN
			fbXmlSrvRead.bExecute := FALSE;
			Ejector.Parameters := EjectorParameters;
			nReadIndex := 60;
		END_IF
	60: // read mandrel parameters
		fbXmlSrvRead.sXPath := '/Configuration/Mandrel';
		fbXmlSrvRead.pSymAddr := ADR(MandrelParameters);
		fbXmlSrvRead.cbSymSize := SIZEOF(MandrelParameters);
		fbXmlSrvRead.bExecute := TRUE;
		nReadIndex := 70;
	70: // wait
		IF NOT fbXmlSrvRead.bBusy THEN
			fbXmlSrvRead.bExecute := FALSE;
			Mandrel.Parameters := MandrelParameters;
			nReadIndex := 80;
		END_IF
	80: // done reading parameters
		ReadParameters := TRUE;		
END_CASE

fbXmlSrvRead(
	sNetId:= '', 
	ePath:= E_OpenPath.PATH_GENERIC, 
	nMode:= XMLSRV_SKIPMISSING, 
	sFilePath:= 'C:\Configuration.xml');
END_METHOD

METHOD SaveParameters : BOOL
VAR_INPUT
	Execute	: BOOL;
END_VAR
VAR_INST
	nSaveIndex	: INT;
	rTrig		: R_TRIG;
END_VAR
SaveParameters := FALSE;

rTrig(CLK := Execute);
IF rTrig.Q THEN
	nSaveIndex := 10;
END_IF

IF NOT Execute THEN
	nSaveIndex := 0;
END_IF

CASE nSaveIndex OF
	10: // read the info from the config file for the camera
		fbXmlSrvWrite.sXPath := '/Configuration/Camera';
		CameraParameters := Camera.Parameters;
		fbXmlSrvWrite.pSymAddr := ADR(CameraParameters);
		fbXmlSrvWrite.cbSymSize := SIZEOF(CameraParameters);
		fbXmlSrvWrite.bExecute := TRUE;
		nSaveIndex := 20;
	20: // wait for the info to load
		IF NOT fbXmlSrvWrite.bBusy THEN
			fbXmlSrvWrite.bExecute := FALSE;
			nSaveIndex := 30;
		END_IF
	30: // read the info from the config file for the cutter
		fbXmlSrvWrite.sXPath := '/Configuration/Cutter';
		CutterParameters := Cutter.Parameters;
		fbXmlSrvWrite.pSymAddr := ADR(CutterParameters);
		fbXmlSrvWrite.cbSymSize := SIZEOF(CutterParameters);
		fbXmlSrvWrite.bExecute := TRUE;
		nSaveIndex := 40;
	40: // wait to complete
		IF NOT fbXmlSrvWrite.bBusy THEN
			fbXmlSrvWrite.bExecute := FALSE;
			nSaveIndex := 50;
		END_IF
	50: // read the ejector parameters
		fbXmlSrvWrite.sXPath := '/Configuration/Ejector';
		EjectorParameters := Ejector.Parameters;
		fbXmlSrvWrite.pSymAddr := ADR(EjectorParameters);
		fbXmlSrvWrite.cbSymSize := SIZEOF(EjectorParameters);
		fbXmlSrvWrite.bExecute := TRUE;
		nSaveIndex := 60;
	60: // wait
		IF NOT fbXmlSrvWrite.bBusy THEN
			fbXmlSrvWrite.bExecute := FALSE;
			nSaveIndex := 70;
		END_IF
	70: // write mandrel parameters
		fbXmlSrvWrite.sXPath := '/Configuration/Mandrel';
		MandrelParameters := Mandrel.Parameters;
		fbXmlSrvWrite.pSymAddr := ADR(MandrelParameters);
		fbXmlSrvWrite.cbSymSize := SIZEOF(MandrelParameters);
		fbXmlSrvWrite.bExecute := TRUE;
		nSaveIndex := 80;
	80: // wait
		IF NOT fbXmlSrvWrite.bBusy THEN
			fbXmlSrvWrite.bExecute := FALSE;
			fbMessageSaved.Send(0);
			nSaveIndex := 90;
		END_IF
	90: // done writing parameters
		SaveParameters := TRUE;		
END_CASE

fbXmlSrvWrite(
	sNetId:= '', 
	ePath:= E_OpenPath.PATH_GENERIC, 
	nMode:= XMLSRV_SKIPMISSING, 
	sFilePath:= 'C:\Configuration.xml');
END_METHOD

END_FUNCTION_BLOCK

// ---- POUs/FB_Base.TcPOU
FUNCTION_BLOCK FB_Base IMPLEMENTS I_UnitState
VAR_INPUT
	eCommand			: Tc3_PackML_V2.E_PMLCommand;
	eModeCommand		: DINT;
END_VAR
VAR_OUTPUT
	eState				: Tc3_PackML_V2.E_PMLState;	
	sState				: STRING;		
	eMode				: DINT;	
END_VAR
VAR
	nState				: INT;
	nClearingState		: INT;
	rTrig				: R_TRIG;
	ePreviousState		: Tc3_PackML_V2.E_PMLState;
	fbStateMachine		: Tc3_PackML_V2.PML_StateMachine;
	fbUnitModeConfig	: Tc3_PackML_V2.PML_UnitModeConfig;
	fbUnitModeManager	: Tc3_PackML_V2.PML_UnitModeManager;
END_VAR

fbStateMachine(
	eMode := eMode,
	eCommand := eCommand,
	eState => eState,
	sState => sState);

// control the mode of the PackML state machine 
// e.g. production, manual, maintenance)
fbUnitModeManager(
	bExecute := (eMode <> eModeCommand),
	eModeCommand := eModeCommand,
	eState := eState,
	eModeStatus => eMode);
IF fbUnitModeManager.bError THEN
	fbUnitModeManager(bExecute := FALSE);
END_IF

// all the case statement in each PackML method use the same index
// this index is reset to zero when the PackML state changes
IF ePreviousState <> eState THEN
	ePreviousState := eState;
	nState := 0;
	nClearingState := 0;
END_IF

// execute PackML method based on PackML state
CASE eState OF
	ePMLState_Undefined: M_Undefined();
	ePMLState_Clearing: M_Clearing();
	ePMLState_Stopped: M_Stopped();
	ePMLState_Starting: M_Starting();
	ePMLState_Idle: M_Idle();
	ePMLState_Suspended: M_Suspended();
	ePMLState_Execute: M_Execute();
	ePMLState_Stopping: M_Stopping();
	ePMLState_Aborting: M_Aborting();
	ePMLSTate_Aborted: M_Aborted();
	ePMLState_Holding: M_Holding();
	ePMLState_Held: M_Held();
	ePMLState_Unholding: M_Unholding();
	ePMLState_Suspending: M_Suspending();
	ePMLState_Unsuspending: M_Unsuspending();
	ePMLState_Resetting: M_Resetting();
	ePMLState_Completing: M_Completing();
	ePMLState_Complete: M_Complete();
END_CASE


METHOD M_Aborted
END_METHOD


METHOD M_Aborting
END_METHOD


METHOD M_Clearing
END_METHOD


METHOD M_Complete
END_METHOD


METHOD M_Completing
END_METHOD


METHOD M_Execute
END_METHOD


METHOD M_Held
END_METHOD


METHOD M_Holding
END_METHOD


METHOD M_Idle
END_METHOD


METHOD M_Resetting
END_METHOD


METHOD M_Starting
END_METHOD

METHOD M_StateComplete
fbStateMachine.M_StateComplete();
END_METHOD


METHOD M_Stopped
END_METHOD


METHOD M_Stopping
END_METHOD


METHOD M_Suspended
END_METHOD


METHOD M_Suspending
END_METHOD


METHOD M_Undefined
END_METHOD


METHOD M_Unholding
END_METHOD


METHOD M_Unsuspending
END_METHOD

END_FUNCTION_BLOCK

// ---- POUs/FB_Mandrel.TcPOU
FUNCTION_BLOCK FB_Mandrel
VAR_INPUT
END_VAR
VAR_OUTPUT
END_VAR
VAR
	// I/O
	Yaxis					: AXIS_REF;			// main axis that goes into and out
	Xaxis					: AXIS_REF;			// cross axis that goes left and right
	Spindle					: AXIS_REF; 		// rotational axis
	VacAxis					: FB_Axis;
	ModeOfOp	AT %Q*		: SINT := 8;		// required by the stepper motor module 
	doVacuum	AT %Q*		: BOOL;				// turns the vacuum on/off
	doStripperExtend AT %Q*	: BOOL;				// actuates the stripper plate
	doStripperRetract AT %Q*: BOOL;
	diVacuumSensor AT %I*	: BOOL;
	aoVacuumSenosr AT %I*	: INT;
	// motion fb's
	mcMoveAbsY				: MC_MoveAbsolute;
	mcMoveRelY				: MC_MoveRelative;
	mcMoveAbsX				: MC_MoveAbsolute;
	mcMoveRelX				: MC_MoveRelative;
	mcMoveRelSpindle		: MC_MoveRelative;
	mcPowerY				: MC_Power;
	mcPowerX				: MC_Power;
	mcPowerSpindle			: MC_Power;
	mcResetX				: MC_Reset;
	mcResetY				: MC_Reset;
	mcResetSpindle			: MC_Reset;
	
// variables in methods
	LiftSampleTon			: TON := (PT := T#500MS);
	LowerSampleTon			: TON := (PT := T#500MS);
	
	_SpindleIncrement		: LREAL;
	_tubeParameters			: ST_TubeParameters;
	_vacuum_mmHg			: REAL;	
	_hmiParameters			: ST_MandrelParameters;
	_parameters				: ST_MandrelParameters;
	fbMessageChange			: FB_TcMessage;
	fbMessageLoaded			: FB_TcMessage;

END_VAR

METHOD Abort : BOOL
VAR_INPUT
END_VAR
DisableSpindle();
DisableX();
DisableY();
VacAxis.Disable();
doStripperExtend := FALSE;
doStripperRetract := FALSE;
MandrelVacuum := FALSE;
END_METHOD

METHOD Clear : INT
VAR_INPUT
	Execute	: BOOL;
END_VAR
VAR_INST
	rTrig	: R_TRIG;
	nIndex	: INT;
END_VAR
rTrig(CLK := Execute);
IF rTrig.Q THEN
	nIndex := 10;
	Reset(Execute := FALSE);
	MoveToLoadPosition(Execute := FALSE);
	VacAxis.AbsMove(Execute := FALSE, Position := 0, Velocity := 0);
END_IF

IF NOT Execute THEN
	nIndex := 0;
END_IF

CASE nIndex OF
	0: // idle state
		Clear := 0;
	10: // reset the mandrel
		IF Reset(Execute := TRUE) = 1 THEN
			Reset(Execute := FALSE);
			nIndex := 20;
		END_IF
	20: // lower the sample
		IF LowerSample() = 1 THEN
			nIndex := 30;
		END_IF
	30: // move to load position
		IF MoveToLoadPosition(Execute := TRUE) = 1 THEN
			MoveToLoadPosition(Execute := FALSE);
			nIndex := 40;
		END_IF
	40: // move the vacuum axis to the vacuum position
		IF VacAxis.AbsMove(Execute := TRUE, Position := _tubeParameters.VacPosition, Velocity := VacuumVelocity) = 1 THEN
			VacAxis.AbsMove(Execute := FALSE, Position := 0, Velocity := 0);
			nIndex := 50;
		END_IF
	50: // done state
		Clear := 1; 
END_CASE
END_METHOD

METHOD ConvertVaccum : BOOL
VAR_INPUT
END_VAR
VAR_INST
	VacuumSensorV	: REAL;
END_VAR
VAR
	VacuumSlope		: REAL;
END_VAR
VacuumSensorV := INT_TO_REAL(aoVacuumSenosr) * 10 / 32767.0;
(* 1V = 0 mmHg, 5V = 760 mmHg *)
VacuumSlope := 760 / 4.0;
_vacuum_mmHg := VacuumSlope * VacuumSensorV - VacuumSlope;
END_METHOD

METHOD DisableSpindle : BOOL
VAR_INPUT
END_VAR
mcPowerSpindle(Axis := Spindle, Enable := FALSE);
Spindle.ReadStatus();
DisableSpindle := NOT Spindle.Status.Operational;
END_METHOD

METHOD DisableX : BOOL
VAR_INPUT
END_VAR
mcPowerX(Axis := XAxis, Enable := FALSE);
XAxis.ReadStatus();
DisableX := NOT XAxis.Status.Operational;
END_METHOD

METHOD DisableY : BOOL
VAR_INPUT
END_VAR
mcPowerY(Axis := YAxis, Enable := FALSE);
YAxis.ReadStatus();
DisableY := NOT YAxis.Status.Operational;
END_METHOD

METHOD EnableSpindle : BOOL
VAR_INPUT
END_VAR
mcPowerSpindle(
	Axis := Spindle, 
	Enable := TRUE,
	Enable_Positive := TRUE,
	Enable_Negative := TRUE);
Spindle.ReadStatus();
EnableSpindle := Spindle.Status.Operational;
END_METHOD

METHOD EnableX : BOOL
VAR_INPUT
END_VAR
mcPowerX(
	Axis := XAxis, 
	Enable := TRUE,
	Enable_Positive := TRUE,
	Enable_Negative := TRUE);
XAxis.ReadStatus();
EnableX := XAxis.Status.Operational;
END_METHOD

METHOD EnableY : BOOL
VAR_INPUT
END_VAR
mcPowerY(
	Axis := YAxis, 
	Enable := TRUE,
	Enable_Positive := TRUE,
	Enable_Negative := TRUE);
YAxis.ReadStatus();
EnableY := YAxis.Status.Operational;
END_METHOD

METHOD FB_init : BOOL
VAR_INPUT
	bInitRetains : BOOL; // if TRUE, the retain variables are initialized (warm start / cold start)
	bInCopyCode : BOOL;  // if TRUE, the instance afterwards gets moved into the copy code (online change)
END_VAR
IF NOT fbMessageChange.EqualsToEventEntryEx(stOther := TC_EVENTS.SlitterEvents.ParameterChange) THEN
	fbMessageChange.CreateEx(TC_EVENTS.SlitterEvents.ParameterChange, 0);
	fbMessageChange.ipArguments.Clear();
END_IF

IF NOT fbMessageLoaded.EqualsToEventEntryEx(stOther := TC_EVENTS.SlitterEvents.ParametersLoadedFromFile) THEN
	fbMessageLoaded.CreateEx(TC_EVENTS.SlitterEvents.ParametersLoadedFromFile, 0);
	fbMessageLoaded.ipArguments.Clear().AddString('Mandrel');
END_IF
END_METHOD

METHOD LiftSample : INT
VAR_INPUT
END_VAR
VAR_INST
END_VAR
doStripperExtend := TRUE;
doStripperRetract := FALSE;
LiftSample := 0;
LiftSampleTon(IN := TRUE);
IF LiftSampleTon.Q THEN
	LiftSample := 1;
	LiftSampleTon(IN := FALSE);
END_IF
END_METHOD

PROPERTY loadPositionX : LREAL
GET
loadPositionX := _parameters.loadPositionX;
END_GET
SET
fbMessageChange.ipArguments.Clear().AddString('loadPositionX').AddLReal(_parameters.loadPositionX).AddLReal(loadPositionX);
fbMessageChange.Send(0);
_parameters.loadPositionX := loadPositionX;
END_SET
END_PROPERTY

PROPERTY loadPositionY : LREAL
GET
loadPositionY := _parameters.loadPositionY;
END_GET
SET
fbMessageChange.ipArguments.Clear().AddString('loadPositionY').AddLReal(_parameters.loadPositionY).AddLReal(loadPositionY);
fbMessageChange.Send(0);
_parameters.loadPositionY := loadPositionY;
END_SET
END_PROPERTY

METHOD LowerSample : INT
VAR_INPUT
END_VAR
doStripperExtend := FALSE;
doStripperRetract := TRUE;
LowerSample := 0;
LowerSampleTon(IN := TRUE);
IF LowerSampleTon.Q THEN
	LowerSample := 1;
	LowerSampleTon(IN := FALSE);
	doStripperRetract := FALSE;
END_IF
END_METHOD

PROPERTY MandrelVacuum : BOOL
GET
MandrelVacuum := doVacuum;
END_GET
SET
doVacuum := MandrelVacuum;
END_SET
END_PROPERTY

METHOD MonitorParameters : BOOL
VAR_INPUT
END_VAR
IF _hmiParameters.loadPositionX <> loadPositionX THEN
	loadPositionX := _hmiParameters.loadPositionX;
END_IF

IF _hmiParameters.loadPositionY <> loadPositionY THEN
	loadPositionY := _hmiParameters.loadPositionY;
END_IF

IF _hmiParameters.spindleOffset <> SpindleOffset THEN
	SpindleOffset := _hmiParameters.spindleOffset;
END_IF

IF _hmiParameters.spindleVelocity <> spindleVelocity THEN
	spindleVelocity := _hmiParameters.spindleVelocity;
END_IF

IF _hmiParameters.velocityX <> velocityX THEN
	velocityX := _hmiParameters.velocityX;
END_IF

IF _hmiParameters.velocityY <> velocityY THEN
	velocityY := _hmiParameters.velocityY;
END_IF

IF _hmiParameters.vacuumVelocity <> VacuumVelocity THEN
	VacuumVelocity := _hmiParameters.vacuumVelocity;
END_IF
END_METHOD

METHOD MoveToCutPosition : INT
VAR_INPUT
	Execute	: BOOL;
	CutPositionX : LREAL;
	CutPositionY : LREAL;
END_VAR
VAR_INST
	nIndex	: INT;
	rTrig	: R_TRIG;
END_VAR
rTrig(CLK := Execute);
IF rTrig.Q THEN
	nIndex := 10;
	mcMoveAbsX(Axis := Xaxis, Execute := FALSE);
	mcMoveAbsY(Axis := YAxis, Execute := FALSE);
	mcMoveRelSpindle(Axis := Spindle, Execute := FALSE);
	MoveToCutPosition := 0;
END_IF

IF NOT Execute THEN
	nIndex := 0;
END_IF

CASE nIndex OF
	0: // idle state
		MoveToCutPosition := 0;
	10: // move
		mcMoveAbsX.Execute := TRUE;
		mcMoveAbsX.Position := CutPositionX;
		mcMoveAbsX.Velocity := _parameters.velocityX;
		
		mcMoveAbsY.Execute := TRUE;
		mcMoveAbsY.Position := CutPositionY;
		mcMoveAbsY.Velocity := _parameters.velocityY;
		
		mcMoveRelSpindle.Execute := TRUE;
		mcMoveRelSpindle.Distance := 3.14159;
		mcMoveRelSpindle.Velocity := 20;
		
		IF mcMoveAbsX.Done AND mcMoveAbsY.Done AND mcMoveRelSpindle.Done THEN
			mcMoveAbsX.Execute := FALSE;
			mcMoveAbsY.Execute := FALSE;
			mcMoveRelSpindle.Execute := FALSE;
			nIndex := 20;
		END_IF
		mcMoveAbsX(Axis := XAxis);
		mcMoveAbsY(Axis := YAxis);
		mcMoveRelSpindle(Axis := Spindle);
	20: // done state
		MoveToCutPosition := 1;
	30: // error state
		MoveToCutPosition := -1;	
END_CASE
END_METHOD

METHOD MoveToEjectPosition : INT
VAR_INPUT
	Execute: BOOL;
	EjectPositionX : LREAL;
	EjectPositionY : LREAL;
END_VAR

VAR_INST
	rTrig: R_TRIG;
	nIndex: INT;
END_VAR
rTrig(CLK := Execute);
IF rTrig.Q THEN
	nIndex := 10;
	mcMoveAbsX(Axis := Xaxis, Execute := FALSE);
	mcMoveAbsY(Axis := YAxis, Execute := FALSE);
END_IF

IF NOT Execute THEN
	nIndex := 0;
END_IF

CASE nIndex OF
	0: // idle state
		MoveToEjectPosition := 0;
	10: // move
		mcMoveAbsX.Execute := TRUE;
		mcMoveAbsX.Position := EjectPositionX;
		mcMoveAbsX.Velocity := _parameters.velocityX;
		
		mcMoveAbsY.Execute := TRUE;
		mcMoveAbsY.Position := EjectPositionY;
		mcMoveAbsY.Velocity := _parameters.velocityY;
		
		IF mcMoveAbsX.Done AND mcMoveAbsY.Done THEN
			mcMoveAbsX.Execute := FALSE;
			mcMoveAbsY.Execute := FALSE;
			nIndex := 20;
		END_IF
		IF mcMoveAbsX.Error THEN
			mcMoveAbsX.Execute := FALSE;
			nIndex := 30;
		END_IF
		mcMoveAbsX(Axis := XAxis);
		mcMoveAbsY(Axis := YAxis);
	20: // done state
		MoveToEjectPosition := 1;
	30: // error state
		MoveToEjectPosition := -1;	
END_CASE
END_METHOD

METHOD MoveToInspectPosition : INT
VAR_INPUT
	Execute	: BOOL;
	InspectPositionX : LREAL;
	InspectPositionY : LREAL;
END_VAR
VAR_INST
	rTrig	: R_TRIG;
	nIndex	: INT;
END_VAR
rTrig(CLK := Execute);
IF rTrig.Q THEN
	nIndex := 10;
	mcMoveAbsX(Axis := Xaxis, Execute := FALSE);
	mcMoveAbsY(Axis := YAxis, Execute := FALSE);
	mcMoveRelSpindle(Axis := Spindle, Execute := FALSE);
END_IF

IF NOT Execute THEN
	nIndex := 0;
END_IF

CASE nIndex OF
	0: // idle state
		MoveToInspectPosition := 0;
	10: // move
		mcMoveRelSpindle.Execute := TRUE;
		mcMoveRelSpindle.Distance := _parameters.spindleOffset;
		mcMoveRelSpindle.Velocity := _parameters.spindleVelocity;
		
		mcMoveAbsX.Execute := TRUE;
		mcMoveAbsX.Position := InspectPositionX;
		mcMoveAbsX.Velocity := _parameters.velocityX;
		
		mcMoveAbsY.Execute := TRUE;
		mcMOveAbsY.Position := InspectPositionY;
		mcMoveAbsY.Velocity := _parameters.velocityY;
		
		IF mcMoveAbsX.Done AND mcMoveAbsY.Done AND mcMoveRelSpindle.Done THEN
			mcMoveAbsX.Execute := FALSE;
			mcMoveAbsY.Execute := FALSE;
			mcMoveRelSpindle.Execute := FALSE;
			nIndex := 20;
		END_IF
		IF mcMoveAbsX.Error THEN
			mcMoveAbsX.Execute := FALSE;
			nIndex := 30;
		END_IF
		mcMoveAbsX(Axis := XAxis);
		mcMoveAbsY(Axis := YAxis);
		mcMoveRelSpindle(Axis := Spindle);
	20: // done state
		MoveToInspectPosition := 1;
	30: // error state
		MoveToInspectPosition := -1;	
END_CASE
END_METHOD

METHOD MoveToLoadPosition : INT
VAR_INPUT
	Execute: BOOL;
END_VAR

VAR_INST
	rTrig: R_TRIG;
	nIndex: INT;
	debug : INT;
END_VAR
rTrig(CLK := Execute);
IF rTrig.Q THEN
	nIndex := 10;
	mcMoveAbsX(Axis := Xaxis, Execute := FALSE);
	mcMoveAbsY(Axis := YAxis, Execute := FALSE);
END_IF

IF NOT Execute THEN
	debug := debug + 1;
	nIndex := 0;
END_IF

CASE nIndex OF
	0: // idle state
		MoveToLoadPosition := 0;
	10: // move
		mcMoveAbsX.Execute := TRUE;
		mcMoveAbsX.Position := _parameters.loadPositionX;
		mcMoveAbsX.Velocity := _parameters.velocityX;
		
		mcMoveAbsY.Execute := TRUE;
		mcMoveAbsY.Position := _parameters.loadPositionY;
		mcMoveAbsY.Velocity := _parameters.velocityY;
		
		IF mcMoveAbsX.Done AND mcMoveAbsY.Done THEN
			mcMoveAbsX.Execute := FALSE;
			mcMoveAbsY.Execute := FALSE;
			nIndex := 20;
		END_IF
		IF mcMoveAbsX.Error THEN
			mcMoveAbsX.Execute := FALSE;
			nIndex := 30;
		END_IF
		mcMoveAbsX(Axis := XAxis);
		mcMoveAbsY(Axis := YAxis);
	20: // done state
		MoveToLoadPosition := 1;
		doStripperRetract := FALSE;
	30: // error state
		MoveToLoadPosition := -1;	
		doStripperRetract := FALSE;
END_CASE
END_METHOD

METHOD MoveToVacPosition : BOOL
VAR_INPUT
	Execute	: BOOL;
END_VAR
VAR_INST
	rTrig	: R_TRIG;
	nIndex	: INT;
END_VAR
MoveToVacPosition := FALSE;

rTrig(CLK := Execute);
IF rTrig.Q THEN
	nIndex := 10;
	VacAxis.AbsMove(Execute := FALSE, Position := 0, Velocity := 0);
END_IF

IF NOT Execute THEN
	nIndex := 0;
END_IF

CASE nIndex OF
	10: // move to location
		IF VacAxis.AbsMove(Execute := TRUE, Position := _tubeParameters.VacPosition, Velocity := _parameters.vacuumVelocity) = 1 THEN
			VacAxis.AbsMove(Execute := FALSE, Position := 0, Velocity := 0);
			nIndex := 20;
		END_IF
	20: // 
		MoveToVacPosition := TRUE;
END_CASE
END_METHOD

METHOD MoveXAbs : INT
VAR_INPUT
	Execute 	: BOOL;
	Position	: LREAL;
END_VAR
VAR_INST
	rTrig	: R_TRIG;
	nIndex	: INT;
END_VAR
rTrig(CLK := Execute);
IF rTrig.Q THEN
	nIndex := 10;
	mcMoveAbsX(Axis := Xaxis, Execute := FALSE);
END_IF

IF NOT Execute THEN
	nIndex := 0;
END_IF

CASE nIndex OF 
	0: // idle state
		MoveXAbs := 0;
	10: // move x axis
		mcMoveAbsX.Execute := TRUE;
		mcMoveAbsX.Position := Position;
		mcMoveAbsX.Velocity := _parameters.velocityX;
		IF mcMoveAbsX.Done THEN
			mcMoveAbsX.Execute := FALSE;
			nIndex := 20;
		END_IF
		IF mcMoveAbsx.Error THEN
			mcMoveAbsX.Execute := FALSE;
			nIndex := 30;
		END_IF
		mcMoveAbsX(Axis := Xaxis);
	20: // done state
		MoveXAbs := 1;
	30: // error state
		MoveXAbs := -1;
END_CASE
END_METHOD

METHOD MoveXRel : INT
VAR_INPUT
	Execute 	: BOOL;
	Distance	: LREAL;
END_VAR
VAR_INST
	rTrig	: R_TRIG;
	nIndex	: INT;
END_VAR
rTrig(CLK := Execute);
IF rTrig.Q THEN
	nIndex := 10;
	mcMoveRelX(Axis := Xaxis, Execute := FALSE);
END_IF

IF NOT Execute THEN
	nIndex := 0;
END_IF

CASE nIndex OF 
	0: // idle state
		MoveXRel := 0;
	10: // move x axis
		mcMoveRelX.Execute := TRUE;
		mcMoveRelX.Distance := Distance;
		mcMoveRelX.Velocity := _parameters.velocityX;
		IF mcMoveRelX.Done THEN
			mcMoveRelX.Execute := FALSE;
			nIndex := 20;
		END_IF
		IF mcMoveRelX.Error THEN
			mcMoveRelX.Execute := FALSE;
			nIndex := 30;
		END_IF
		mcMoveRelX(Axis := Xaxis);
	20: // done state
		MoveXRel := 1;
	30: // error state
		MoveXRel := -1;
END_CASE
END_METHOD

METHOD MoveYAbs : INT
VAR_INPUT
	Execute		: BOOL;
	Position	: LREAL;
END_VAR

VAR_INST
	rTrig		: R_TRIG;
	nIndex		: INT;
END_VAR
rTrig(CLK := Execute);
IF rTrig.Q THEN
	nIndex := 10;
	mcMoveAbsY(Axis := Yaxis, Execute := FALSE);
END_IF

IF NOT Execute THEN
	nIndex := 0;
END_IF

CASE nIndex OF 
	0: // idle state
		MoveYAbs := 0;
	10: // move x axis
		mcMoveAbsY.Execute := TRUE;
		mcMoveAbsY.Position := Position;
		mcMoveAbsY.Velocity := _parameters.velocityY;
		IF mcMoveAbsY.Done THEN
			mcMoveAbsY.Execute := FALSE;
			nIndex := 20;
		END_IF
		IF mcMoveAbsY.Error THEN
			mcMoveAbsY.Execute := FALSE;
			nIndex := 30;
		END_IF
		mcMoveAbsY(Axis := Yaxis);
	20: // done state
		MoveYAbs := 1;
	30: // error state
		MoveYAbs := -1;
END_CASE
END_METHOD

METHOD MoveYRel : INT
VAR_INPUT
	Execute 	: BOOL;
	Distance	: LREAL;
END_VAR
VAR_INST
	rTrig	: R_TRIG;
	nIndex	: INT;
END_VAR
rTrig(CLK := Execute);
IF rTrig.Q THEN
	nIndex := 10;
	mcMoveRelY(Axis := Yaxis, Execute := FALSE);
END_IF

IF NOT Execute THEN
	nIndex := 0;
END_IF

CASE nIndex OF 
	0: // idle state
		MoveYRel := 0;
	10: // move x axis
		mcMoveRelY.Execute := TRUE;
		mcMoveRelY.Distance := Distance;
		mcMoveRelY.Velocity := _parameters.velocityY;
		IF mcMoveRelY.Done THEN
			mcMoveRelY.Execute := FALSE;
			nIndex := 20;
		END_IF
		IF mcMoveRelY.Error THEN
			mcMoveRelY.Execute := FALSE;
			nIndex := 30;
		END_IF
		mcMoveRelY(Axis := Yaxis);
	20: // done state
		MoveYRel := 1;
	30: // error state
		MoveYRel := -1;
END_CASE
END_METHOD

PROPERTY OperationalSpindle : BOOL
GET
Spindle.ReadStatus();
OperationalSpindle := Spindle.Status.Operational;
END_GET
END_PROPERTY

PROPERTY OperationalX : BOOL
GET
XAxis.ReadStatus();
OperationalX := XAxis.Status.Operational;
END_GET
END_PROPERTY

PROPERTY OperationalY : BOOL
GET
YAxis.ReadStatus();
OperationalY := YAxis.Status.Operational;
END_GET
END_PROPERTY

PROPERTY Parameters : ST_MandrelParameters
GET
Parameters := _parameters;
END_GET
SET
fbMessageLoaded.Send(0);
_parameters := Parameters;
_hmiParameters := Parameters;
END_SET
END_PROPERTY

METHOD Reset : INT
VAR_INPUT
	Execute	: BOOL;
END_VAR
VAR_INST
	nIndex 	: INT;
	rTrig	: R_TRIG;
END_VAR
rTrig(CLK := Execute);
IF rTrig.Q THEN
	nIndex := 10;
	LiftSampleTon(IN := FALSE);
	LowerSampleTon(IN := FALSE);
	VacAxis.Reset(Execute := FALSE);
END_IF

IF NOT Execute THEN
	nIndex := 0;
END_IF

Xaxis.ReadStatus();
YAxis.ReadStatus();
Spindle.ReadStatus();

CASE nIndex OF
	0:// idle state
		Reset := 0;
	10: // check if there are any errors on the drives
		IF XAxis.Status.Error THEN
			nIndex := 20;
		ELSIF YAxis.Status.Error THEN
			nIndex := 30;
		ELSIF Spindle.Status.Error THEN
			nIndex := 40;
		ELSIF VacAxis.Error THEN
			nIndex := 45;
		ELSE
			nIndex := 50;
		END_IF
	20: // reset x axis
		mcResetX.Execute := TRUE;
		IF mcResetX.Done THEN
			nIndex := 10;
			mcResetX.Execute := FALSE;
		END_IF
		mcResetX(Axis := XAxis);
	30: // reset y axis
		mcResetY.Execute := TRUE;
		IF mcResetY.Done THEN
			nIndex := 10;
			mcResetY.Execute := FALSE;
		END_IF
		mcResetY(Axis := YAxis);
	40: // reset spindle axis
		mcResetSpindle.Execute := TRUE;
		IF mcResetSpindle.Done THEN
			nIndex := 10;
			mcResetSpindle.Execute := FALSE;
		END_IF
		mcResetSpindle(Axis := Spindle);
	45: // reset the vac axis
		
		IF VacAxis.Reset(Execute := TRUE) THEN
			VacAxis.Reset(Execute := FALSE);
			nIndex := 10;
		END_IF
		
	50: // enable the drives
		mcPowerX(Axis := XAxis, Enable := TRUE, Enable_Negative := TRUE, Enable_Positive := TRUE);
		mcPowerY(Axis := YAxis, Enable := TRUE, Enable_Negative := TRUE, Enable_Positive := TRUE);
		mcPowerSpindle(Axis := Spindle, Enable := TRUE, Enable_Negative := TRUE, Enable_Positive := TRUE);
		IF XAxis.Status.Operational 
			AND YAxis.Status.Operational 
			AND Spindle.Status.Operational 
			AND VacAxis.Enable() THEN
				nIndex := 60;
		END_IF
	60: // done state
		Reset := 1;			
END_CASE
END_METHOD

METHOD RotateSpindle : INT
VAR_INPUT
	Execute : BOOL;
	Distance	: LREAL;
END_VAR
VAR_INST
	nIndex : INT;
	rTrig	: R_TRIG;
END_VAR
rTrig(CLK := Execute);
IF rTrig.Q THEN
	nIndex := 10;
	mcMoveRelSpindle(Axis := Spindle, Execute := FALSE);
END_IF

IF NOT Execute THEN
	nIndex := 0;
END_IF

CASE nIndex OF
	0: // idle state
		RotateSpindle := 0;
	10: // move relative
		mcMoveRelSpindle.Execute := TRUE;
		mcMoveRelSpindle.Distance := Distance;
		mcMoveRelSpindle.Velocity := _parameters.spindleVelocity;
		IF mcMoveRelSpindle.Done THEN
			mcMoveRelSpindle.Execute := FALSE;
			nIndex := 20;
		END_IF
		IF mcMoveRelSpindle.Error THEN
			mcMoveRelSpindle.Execute := FALSE;
			nIndex := 30;
		END_IF
		mcMoveRelSpindle(Axis := Spindle);
	20: // done state
		RotateSpindle := 1;
	30: // error state
		RotateSpindle := -1;
END_CASE
END_METHOD

PROPERTY SpindleIncrement : LREAL
GET
SpindleIncrement := _spindleIncrement;
END_GET
SET
_SpindleIncrement := SpindleIncrement;
END_SET
END_PROPERTY

PROPERTY SpindleOffset : LREAL
GET
SpindleOffset := _parameters.spindleOffset;
END_GET
SET
fbMessageChange.ipArguments.Clear().AddString('SpindleOffset').AddLReal(_parameters.spindleOffset).AddLReal(SpindleOffset);
fbMessageChange.Send(0);
_parameters.spindleOffset := SpindleOffset;
END_SET
END_PROPERTY

PROPERTY spindleVelocity : LREAL
GET
spindleVelocity := _parameters.spindleVelocity;
END_GET
SET
fbMessageChange.ipArguments.Clear().AddString('spindleVelocity').AddLReal(_parameters.spindleVelocity).AddLReal(spindleVelocity);
fbMessageChange.Send(0);
_parameters.spindleVelocity := spindleVelocity;
END_SET
END_PROPERTY

PROPERTY TubeParameters : ST_TubeParameters
GET
TubeParameters := _tubeParameters;
END_GET
SET
_tubeParameters := TubeParameters;
END_SET
END_PROPERTY

PROPERTY VacuumSensor : REAL
GET
VacuumSensor := _vacuum_mmHg;
END_GET
END_PROPERTY

PROPERTY VacuumVelocity : LREAL
GET
VacuumVelocity := _parameters.vacuumVelocity;
END_GET
SET
fbMessageChange.ipArguments.Clear().AddString('VacuumVelocity').AddLReal(_parameters.vacuumVelocity).AddLReal(VacuumVelocity);
fbMessageChange.Send(0);
_parameters.vacuumVelocity := VacuumVelocity;
END_SET
END_PROPERTY

PROPERTY velocityX : LREAL
GET
velocityX := _parameters.velocityX;
END_GET
SET
fbMessageChange.ipArguments.Clear().AddString('velocityX').AddLReal(_parameters.velocityX).AddLReal(velocityX);
fbMessageChange.Send(0);
_parameters.velocityX := velocityX;
END_SET
END_PROPERTY

PROPERTY velocityY : LREAL
GET
velocityY := _parameters.velocityY;
END_GET
SET
fbMessageChange.ipArguments.Clear().AddString('velocityY').AddLReal(_parameters.velocityY).AddLReal(velocityY);
fbMessageChange.Send(0);
_parameters.velocityY := velocityY;
END_SET
END_PROPERTY

END_FUNCTION_BLOCK

// ---- POUs/FB_Axis.TcPOU
FUNCTION_BLOCK FB_Axis
VAR_INPUT
END_VAR
VAR_OUTPUT
END_VAR
VAR
	axis	: AXIS_REF;
	mcPower	: MC_Power;
	mcMove	: MC_MoveAbsolute;
	mcReset	: MC_Reset;
	fbAlarm	: FB_TcAlarm;
	
	_error	: BOOL;
	_errorId	: UDINT;
END_VAR

METHOD AbsMove : BOOL
VAR_INPUT
	Execute	: BOOL;
	Position	: LREAL;
	Velocity	: LREAL;
END_VAR
VAR_INST
	nState	: INT;
	rTrig	: R_TRIG;
END_VAR
AbsMove := FALSE;

rTrig(Clk := Execute);
IF rTrig.Q THEN
	nState := 10;
	mcMove(Axis := Axis, Execute := FALSE);
END_IF

IF NOT Execute THEN
	nState := 0;
END_IF

CASE nState OF
	10: // move
		mcMove.Position := Position;
		mcMove.Velocity := Velocity;
		mcMove.Execute := TRUE;
		IF McMove.Done THEN
			nState := 20;
			mcMove.Execute := FALSE;
		END_IF
		IF mcMove.Error THEN
			_error := TRUE;
			_errorId := mcMove.ErrorID;
			fbAlarm.ipArguments.Clear().AddUDInt(_errorId);
			fbAlarm.Raise(0);
			mcMove.Execute := FALSE;
			nState := 20;
		END_IF
		mcMove(Axis := Axis);
	20: // done state
		AbsMove := TRUE;
END_CASE
END_METHOD

METHOD Disable : BOOL
VAR_INPUT
END_VAR
Axis.ReadStatus();
Disable := NOT mcPower.Status;
mcPower(Axis := Axis, Enable := FALSE);
END_METHOD

METHOD Enable : BOOL
VAR_INPUT
END_VAR
axis.ReadStatus();
Enable := mcPower.Status AND axis.Status.Operational;
mcPower(axis := axis, enable := TRUE, Enable_Positive := TRUE, Enable_Negative := TRUE);
END_METHOD

PROPERTY Error : BOOL
GET
Error := Axis.NcToPlc.ErrorCode <> 0 OR _error;
END_GET
END_PROPERTY

METHOD FB_init : BOOL
VAR_INPUT
	bInitRetains : BOOL; // if TRUE, the retain variables are initialized (warm start / cold start)
	bInCopyCode : BOOL;  // if TRUE, the instance afterwards gets moved into the copy code (online change)
END_VAR
IF fbAlarm.EqualsToEventEntryEx(stOther := TC_EVENTS.SlitterEvents.EjectorAxisError) THEN
	fbAlarm.CreateEx(TC_EVENTS.SlitterEvents.EjectorAxisError, FALSE, 0);
	fbAlarm.ipArguments.Clear();
END_IF
END_METHOD

PROPERTY IsEnabled : BOOL
GET
Axis.ReadStatus();
IsEnabled := mcPower.Status AND Axis.Status.Operational;
END_GET
END_PROPERTY

METHOD Reset : BOOL
VAR_INPUT
	Execute : BOOL;
END_VAR
VAR_INST
	nState	: INT;
	rTrig	: R_TRIG;
END_VAR
Reset := FALSE;
rTrig(CLK := Execute);
IF rTrig.Q THEN
	mcMove(Axis := Axis, Execute := FALSE);
	mcReset(Axis := Axis, Execute := FALSE);
	_error := FALSE;
	_errorId := 0;
	nState := 10;
END_IF
IF NOT Execute THEN
	nState := 0;
END_IF
CASE nState OF
	10: // reset the system
		IF fbAlarm.bRaised THEN
			fbAlarm.Clear(0, FALSE);
		END_IF
		mcReset.Execute := TRUE;
		IF mcReset.Done THEN
			mcReset.Execute := FALSE;
			nState := 20;
		END_IF
		IF mcReset.Error THEN
			_error := TRUE;
			_errorId := mcReset.ErrorID;
			fbAlarm.ipArguments.Clear().AddUDInt(_errorId);
			fbAlarm.Raise(0);
			nState := 20;
		END_IF
		mcReset(Axis := Axis);
	20: // done state
		Reset := TRUE;
END_CASE
END_METHOD

END_FUNCTION_BLOCK

// ---- POUs/FB_Camera.TcPOU
FUNCTION_BLOCK FB_Camera
VAR_INPUT
END_VAR
VAR_OUTPUT
END_VAR
VAR
	Trigger	AT %Q*			: BOOL;				// signal to take picture and analyze
	CameraData				: ST_CameraData;	// modbus camera data
	VisionStatus			: ARRAY[0..3] OF BYTE;// modbus camera status
	_tubeParameters			: ST_TubeParameters;
	_pass					: BOOL;
	_fail					: BOOL;
	_noDetect				: BOOL;
			
	_xPoints 				: ARRAY[1..GVL.NumberVisionPoints] OF LREAL;
	_yPoints 				: ARRAY[1..GVL.NumberVisionPoints] OF LREAL;
	_xEllipsePoints			: ARRAY[1..GVL.NumberEllipsePoints] OF LREAL;
	_yEllipsePoints			: ARRAY[1..GVL.NumberEllipsePoints] OF LREAL;
		
	_displayVisionPts		: ARRAY[1..2,1..GVL.NumberVisionPoints] OF LREAL;
	_displayEllipsePts		: ARRAY[1..2,1..GVL.NumberEllipsePoints] OF LREAL;
	_columnPeak				: LREAL;	// xPeak value of the vision points
	_rowPeak				: LREAL;	// yPeak value of the vision points
	_rowCenterLine			: LREAL;	// based on entered minor value -> y value at the center-line axis
	_minorCalculated 		: LREAL;
	_majorCalculated		: LREAL;
	_xEllipseCenter			: LREAL;
	_yEllipseCenter			: LREAL;

	(* for calculating the pitch *)	
	_patternX1				: LREAL;
	_patternX2				: LREAL;
	_patternX3				: LREAL;
	_patternY1				: LREAL;
	_patternY2				: LREAL;
	_patternY3				: LREAL;
	
	(* calculation variables *)
	DeltaXpx				: LREAL;	// distance from peak of curve to center of cut (row)
	DeltaYpx				: LREAL;	// distance from peak of curve to center of cut (column)
	CutLength				: LREAL;
	CutHeight				: LREAL;
	DeltaXmm				: LREAL;
	DeltaYmm				: LREAL;
	(* results *)
	_CutLengthWithOffset	: LREAL;
	_DeltaXmmWithOffset		: LREAL;
	_DeltaYmmWithOffset		: LREAL;
	
	_depthOffset			: REAL; 				// difference due to the plane of cut is different than plane of pattern detect
	_minorRadiusMm			: LREAL := 2.5955;		// minor radius of ellipse in mm
	_majorRadiusMm			: LREAL;
	_slitCenterApparentRow	: LREAL;				// [px] this is the center of the part in x when accounting for the offset due to vision plane versus cut plane
	_tubeCenter				: LREAL;
	_tubeCenterOffset		: LREAL;
	_tubeCenterWithOffset	: LREAL;
	_cameraProgram			: STRING;
	_previousTubeIndex		: INT;
	
	_hmiParameters			: ST_CameraParameters;
	_parameters				: ST_CameraParameters;
	fbMessageChange			: FB_TcMessage;
	fbMessageLoaded			: FB_TcMessage;
END_VAR

PROPERTY angle : LREAL
GET
angle := _parameters.angle;
END_GET
SET
fbMessageChange.ipArguments.Clear().AddString('Angle').AddLReal(_parameters.angle).AddLReal(angle);
fbMessageChange.Send(0);
_parameters.angle := angle;
END_SET
END_PROPERTY

METHOD Calibrate : BOOL
VAR_INPUT
END_VAR
_hmiParameters.pitchRow := (CalibrationDistance / ABS(PatternY1 - PatternY2));
_hmiParameters.pitchColumn := (CalibrationDistance / ABS(PatternX2 - PatternX3));
END_METHOD

PROPERTY CalibrationDistance : LREAL
GET
CalibrationDistance := _parameters.calibrationDistance;
END_GET
SET
fbMessageChange.ipArguments.Clear().AddString('Calibration Distance').AddLReal(_parameters.calibrationDistance).AddLReal(CalibrationDistance);
fbMessageChange.Send(0);
_parameters.calibrationDistance := CalibrationDistance;
END_SET
END_PROPERTY

PROPERTY CameraProgram : STRING
GET
CameraProgram := _cameraProgram;
END_GET
SET
_cameraProgram := CameraProgram;
END_SET
END_PROPERTY

METHOD Compute : INT
VAR_INPUT
	Execute		: BOOL;
END_VAR
VAR_INST
	rTrig			: R_TRIG;
	nIndex			: INT;
	fbSecond		: FB_SecondOrder;
 	fbFourth		: FB_FourthOrder;
	fbEllipse		: FB_Ellipse;
	zeroValues		: BOOL;
END_VAR

VAR
	i: INT;
	yValue	: LREAL;
END_VAR
(* when computing the new cut positions, subtract the delta values from the 
original cut positions *)

rTrig(CLK := Execute);
IF rTrig.Q THEN
	nIndex := 10;
END_IF

IF NOT Execute THEN
	nIndex := 0;
END_IF

CASE nIndex OF
	0: // idle state
		Compute := 0;
	10: // get data
		IF GetCameraData() = 1 THEN
			nIndex := 15;
		END_IF
	15: // did pattern match find _xPoints, _yPoints?
		zeroValues := FALSE;
		FOR i := 1 TO GVL.NumberVisionPoints DO
			IF _xPoints[i] = 0 OR _yPoints[i] = 0 THEN
				zeroValues := TRUE;
			END_IF
		END_FOR
		IF zeroValues THEN
			nIndex := 60;
		ELSE
			nIndex := 20;
		END_IF
	20: // compute the peak x value of the data		
		fbSecond.FindPeak(xValues := ADR(_xPoints), yValues := ADR(_yPoints), xPeak := ADR(_columnPeak));
		fbFourth.FindYatX(xValues := ADR(_xPoints), yValues := ADR(_yPoints), xPeak := ADR(_columnPeak), yPeak := ADR(_rowPeak));
		DeltaYpx := CameraData.Results.LocationInX - _columnPeak;
		DeltaYmm := DeltaYpx * _hmiParameters.pitchColumn;
		_DeltaYmmWithOffset := DeltaYmm + _tubeParameters.AdjustmentY;
		
		CutLength := CameraData.Results.WidthMeasurement * _hmiParameters.pitchColumn;		
		_CutLengthWithOffset := CutLength + _tubeParameters.AdjustmentLength;
		CutHeight := CameraData.Results.HeightMeasurement * _hmiParameters.pitchRow;
		
		_tubeCenter := _rowPeak + 0.5*_tubeParameters.Diameter /_hmiParameters.pitchRow;
		_tubeCenterOffset := (_tubeParameters.DepthOfPocket*TAN(_hmiParameters.angle * 2*3.14159/360.0))/_hmiParameters.pitchRow;
		_tubeCenterWithOffset := _tubeCenter + _tubeCenterOffset;
		
		DeltaXpx := (CameraData.Results.LocationInY - 0.5*CameraData.Results.HeightMeasurement) - _tubeCenterWithOffset;
		DeltaXmm := DeltaXpx * _hmiParameters.pitchRow;
		_DeltaXmmWithOffset := DeltaXmm + _tubeParameters.AdjustmentX;
		
		nIndex := 50;
	30: // compute ellipse
		fbEllipse.EllipseFit(xValues := _xEllipsePoints, yValues := _yEllipsePoints);
		nIndex := 40;
		
	40: // assign values
		_minorCalculated := fbEllipse.minor;
		_majorCalculated := fbEllipse.major;
		_xEllipseCenter := fbEllipse.centrex;
		_yEllipseCenter := fbEllipse.centrey;
		nIndex := 50;
	50: // done state
		Compute := 1;		
	60: // didn't find the pattern, so can't compute a peak
		Compute := -1;					
END_CASE
END_METHOD

PROPERTY CutLengthWithOffset : LREAL
GET
CutLengthWithOffset := _CutLengthWithOffset;
END_GET
END_PROPERTY

PROPERTY DeltaXmmWithOffset : LREAL
GET
DeltaXmmWithOffset := _DeltaXmmWithOffset;
END_GET
END_PROPERTY

PROPERTY DeltaYmmWithOffset : LREAL
GET
DeltaYmmWithOffset := _DeltaYmmWithOffset;
END_GET
END_PROPERTY

PROPERTY Fail : BOOL
GET
Fail := _fail;
END_GET
SET
_fail := Fail;
END_SET
END_PROPERTY

METHOD FB_init : BOOL
VAR_INPUT
	bInitRetains : BOOL; // if TRUE, the retain variables are initialized (warm start / cold start)
	bInCopyCode : BOOL;  // if TRUE, the instance afterwards gets moved into the copy code (online change)
END_VAR
IF NOT fbMessageChange.EqualsToEventEntryEx(stOther := TC_EVENTS.SlitterEvents.ParameterChange) THEN
	fbMessageChange.CreateEx(TC_EVENTS.SlitterEvents.ParameterChange, 0);
	fbMessageChange.ipArguments.Clear();
END_IF

IF NOT fbMessageLoaded.EqualsToEventEntryEx(stOther := TC_EVENTS.SlitterEvents.ParametersLoadedFromFile) THEN
	fbMessageLoaded.CreateEx(TC_EVENTS.SlitterEvents.ParametersLoadedFromFile, 0);
	fbMessageLoaded.ipArguments.Clear().AddString('Camera');
END_IF
END_METHOD

METHOD GetCameraData : INT
VAR_INPUT
END_VAR

VAR_INST
	i				: INT;
	fbMBRegRead		: FB_MBReadRegs;
END_VAR
// format on Cognex needs to be little endian 
GetCameraData := 0;
fbMBRegRead.bExecute := TRUE;

fbMBRegRead.sIPAddr := GVL.CameraIpAddress;
fbMBRegRead.nTCPPort := 502;
fbMBRegRead.nUnitID := 16#FF;
fbMBRegRead.nQuantity := 94; // 188/2;
fbMBRegRead.nMBAddr := GVL.ModbusReadOffset+5;
fbMBRegRead.cbLength := SIZEOF(CameraData.Results);
fbMBRegRead.pDestAddr := ADR(CameraData.Results);

fbMBRegRead();

IF NOT fbMBRegRead.bBusy THEN
	IF NOT fbMBRegRead.bError THEN
		fbMBRegRead(bExecute := FALSE);
		FOR i := 1 TO GVL.NumberVisionPoints DO
			_yPoints[i] := REAL_TO_LREAL(CameraData.Results.PointValueRow[i]);
			_xPoints[i] := REAL_TO_LREAL(CameraData.Results.PointValueColumn[i]);
			_displayVisionPts[1,i] := INT_TO_LREAL(LREAL_TO_INT(_xPoints[i]*100))/100.0; // column values
			_displayVisionPts[2,i] := INT_TO_LREAL(LREAL_TO_INT(_yPoints[i]*100))/100.0; // row values	
		END_FOR

		GetCameraData := 1;	
	ELSE
		fbMBRegRead(bExecute := FALSE);
		FOR i := 1 TO GVL.NumberVisionPoints DO
			_xPoints[i] := 0;
			_yPoints[i] := 0;
			_displayVisionPts[1,i] := 0;
			_displayVisionPts[2,i] := 0;
	
		END_FOR
		GetCameraData := -1;	
		
	END_IF
END_IF
END_METHOD

METHOD Inspect : INT
VAR_INPUT
	Execute	: BOOL;
END_VAR
VAR_INST
	nIndex 	: INT;
	rTrig	: R_TRIG;
	CountStart : REAL;
	CountFinish : REAL;
	Count	: REAL;
	CameraTON	: TON := (PT := T#250MS);
	CameraDataResult : INT;
END_VAR
rTrig(CLK := Execute);
IF rTrig.Q THEN
	Inspect := 0;
	nIndex := 10;
	Trigger := FALSE;
	Compute(Execute := FALSE);
	CameraTON(IN := FALSE);
END_IF

IF NOT Execute THEN
	nIndex := 0;
END_IF

